WHILE NOT endMainLoop DO							
	IF left < right THEN                	
		pPivotElement										:= pCompareElement + (SizeOfStruct * TO_UDINT(SHR(right+left,1)));
		i 													:= left -1;
		j 													:= right +1;
		endSubLoop 											:= FALSE;
		REPEAT
			IF SortInverse
			THEN	// sort descending	
				REPEAT	
					i 										:= i+1;	
					pCmpElement								:= pCompareElement + (SizeOfStruct * TO_UDINT(i-1));
					FOR k := 0 TO MAX_WSTRING_LENGTH DO // Find unequal char
						// element 1,2 to upper char 	https://www.uni-due.de/hummell/infos/ascii/
						IF pCmpElement^[k] = 0 
							AND IgnoreBlank
						THEN
							CompareElement					:= 127;
						ELSE
							CompareElement					:= SEL(pCmpElement^[k] >= 97(*a*)	AND_THEN pCmpElement^[k] <= 122(*z*), 	pCmpElement^[k],pCmpElement^[k] - 32);		// a --> A
						END_IF
						IF pPivotElement^[k] = 0 
							AND IgnoreBlank
						THEN
							PivotElement					:= 127;
						ELSE
							PivotElement					:= SEL(pPivotElement^[k] >= 97(*a*) AND_THEN pPivotElement^[k] <= 122(*z*), pPivotElement^[k], 	pPivotElement^[k] - 32);// a --> A
						END_IF
						// Find unequal char
						IF CompareElement <> PivotElement
							OR CompareElement = 0
							OR PivotElement = 0
						THEN
							EXIT;
						END_IF
					END_FOR
				UNTIL (CompareElement <= PivotElement) OR NOT (i < right)	END_REPEAT	
				REPEAT	
					j 										:= j-1;	
					pCmpElement								:= pCompareElement + (SizeOfStruct * TO_UDINT(j-1));
					FOR k := 0 TO MAX_WSTRING_LENGTH DO // Find unequal char
						// element 1,2 to upper char 	https://www.uni-due.de/hummell/infos/ascii/
						IF pCmpElement^[k] = 0 
							AND IgnoreBlank
						THEN
							CompareElement					:= 127;
						ELSE
							CompareElement					:= SEL(pCmpElement^[k] >= 97(*a*)	AND_THEN pCmpElement^[k] <= 122(*z*), 	pCmpElement^[k],pCmpElement^[k] - 32);		// a --> A
						END_IF
						IF pPivotElement^[k] = 0 
							AND IgnoreBlank
						THEN
							PivotElement					:= 127;
						ELSE
							PivotElement					:= SEL(pPivotElement^[k] >= 97(*a*) AND_THEN pPivotElement^[k] <= 122(*z*), pPivotElement^[k], 	pPivotElement^[k] - 32);// a --> A
						END_IF
						// Find unequal char
						IF CompareElement <> PivotElement
							OR CompareElement = 0
							OR PivotElement = 0
						THEN
							EXIT;
						END_IF
					END_FOR
				UNTIL (CompareElement >= PivotElement) OR NOT (j > left)	END_REPEAT		
			ELSE	// sort ascending
				REPEAT	
					i 										:= i+1;
					pCmpElement								:= pCompareElement + (SizeOfStruct * TO_UDINT(i-1));
					FOR k := 0 TO MAX_WSTRING_LENGTH DO // Find unequal char
						// element 1,2 to upper char 	https://www.uni-due.de/hummell/infos/ascii/
						IF pCmpElement^[k] = 0 
							AND IgnoreBlank
						THEN
							CompareElement					:= 127;
						ELSE
							CompareElement					:= SEL(pCmpElement^[k] >= 97(*a*)	AND_THEN pCmpElement^[k] <= 122(*z*), 	pCmpElement^[k],pCmpElement^[k] - 32);		// a --> A
						END_IF
						IF pPivotElement^[k] = 0 
							AND IgnoreBlank
						THEN
							PivotElement					:= 127;
						ELSE
							PivotElement					:= SEL(pPivotElement^[k] >= 97(*a*) AND_THEN pPivotElement^[k] <= 122(*z*), pPivotElement^[k], 	pPivotElement^[k] - 32);// a --> A
						END_IF
						// Find unequal char
						IF CompareElement <> PivotElement
							OR CompareElement = 0
							OR PivotElement = 0
						THEN
							EXIT;
						END_IF
					END_FOR
				UNTIL (CompareElement >= PivotElement)	OR NOT (i < right)	END_REPEAT;				
				REPEAT	
					j 										:= j-1;	
					pCmpElement								:= pCompareElement + (SizeOfStruct * TO_UDINT(j-1));
					FOR k := 0 TO MAX_WSTRING_LENGTH DO // Find unequal char
						// element 1,2 to upper char 	https://www.uni-due.de/hummell/infos/ascii/
						IF pCmpElement^[k] = 0 
							AND IgnoreBlank
						THEN
							CompareElement					:= 127;
						ELSE
							CompareElement					:= SEL(pCmpElement^[k] >= 97(*a*)	AND_THEN pCmpElement^[k] <= 122(*z*), 	pCmpElement^[k],pCmpElement^[k] - 32);		// a --> A
						END_IF
						IF pPivotElement^[k] = 0 
							AND IgnoreBlank
						THEN
							PivotElement					:= 127;
						ELSE
							PivotElement					:= SEL(pPivotElement^[k] >= 97(*a*) AND_THEN pPivotElement^[k] <= 122(*z*), pPivotElement^[k], 	pPivotElement^[k] - 32);// a --> A
						END_IF
						// Find unequal char
						IF CompareElement <> PivotElement
							OR CompareElement = 0
							OR PivotElement = 0
						THEN
							EXIT;
						END_IF
					END_FOR
				UNTIL (CompareElement <= PivotElement) OR NOT (j > left)	END_REPEAT;
			END_IF
			IF i >= j THEN
				endSubLoop									:= TRUE;
			ELSE                    					
				Allocate(SizeOfStruct);
				pElement_1									:= pData + (SizeOfStruct * TO_UDINT(j-1));
				pElement_2									:= pData + (SizeOfStruct * TO_UDINT(i-1));
				
				IF pElement_Tmp = 0 
					OR_ELSE MEMCPY(pElement_Tmp, pElement_1,	SizeOfStruct) = 0
					OR_ELSE MEMCPY(pElement_1,	pElement_2,		SizeOfStruct) = 0
					OR_ELSE MEMCPY(pElement_2,	pElement_Tmp,	SizeOfStruct) = 0
				THEN
					byWSTRING								:= FALSE;
					RETURN;	
				END_IF

			END_IF
		UNTIL endSubLoop END_REPEAT;		
		stack[stackCount] 									:= TO_UDINT(right); 	// save right in stack			
		IF stackCount < 32              					
		THEN                            					
			stackCount 										:= stackCount +1;
		ELSE															// Error stack Limit    
			endMainLoop 									:= TRUE;
			byWSTRING										:= FALSE;			
		END_IF                          					
		right 												:= MAX(left, i-1);
	ELSE                                
		IF stackCount = 1 THEN          
			endMainLoop 									:= TRUE;
		ELSE                            					
			left 											:= right+1;       
			stackCount 										:= stackCount -1;	// load from stack
			right											:= TO_DINT(stack[stackCount]);
		END_IF
	END_IF
END_WHILE
END_METHOD

METHOD FB_exit : BOOL
VAR_INPUT
	bInCopyCode : BOOL; // if TRUE, the exit method is called for exiting an instance that is copied afterwards (online change).
END_VAR
IF NOT bInCopyCode AND pElement_Tmp <> 0
THEN //Release memory in case the PLC stopps
	__DELETE(pElement_Tmp);
END_IF
END_METHOD

END_FUNCTION_BLOCK

// POUs/EventLogger/ReadEvents/EventlogRead
{attribute 'no_check'}
//Read TwinCat ADS evenlogger messages via ADS into PLC in Unicode format
FUNCTION_BLOCK EventlogRead EXTENDS FbBase
VAR CONSTANT
	IGRP_ENUMEVENTS											: UDINT := 16#190;
	IOFFS_ENUM_CONTINUE										: UDINT := 16#1020;
	IOFFS_ENUM_CLOSE										: UDINT := 16#1030;
                                        					
	IGRP_GETTEXT											: UDINT := 16#1F4;
	IOFFS_GETCOMPLETESTRING									: UDINT := 16#0;
	IOFFS_GETSOURCENAME										: UDINT := 16#1;
                                        					
	IOFFS_BEGINENUMACTIVE									: UDINT := 16#0;
	IOFFS_BEGINENUMLOGGED									: UDINT := 16#1;
                                        	
	IGRP_TCEVENTSTREAM_SIMPLE								: UDINT := 16#1;
	IOFFS_TCEVENTCLASS_NONE 								: UDINT := 16#0;
END_VAR
VAR_OUTPUT CONSTANT
	MIN_EVENT												: INT := 1; 
	MAX_EVENT												: INT := PARAM.EVENT_HANDLING_CONFIG.EVENTLOG_READ_MAX_EVENTS ; //End index event list  - see library parameter to customize parameter
	
{attribute 'displaymode':='binary'}
	OPTION_USE_STATE_FOR_TIMESTAMP							: 	BYTE :=2#0000_0001; //option to enable timestamp according to event state instead of only signaled timestamp
{attribute 'displaymode':='binary'}
	OPTION_GET_HOSTNAME_FOR_EACH_EVENT						: 	BYTE :=2#0000_0010; //option to read host name for each single event
END_VAR                                 					
VAR_INPUT                               					
	LangId													: eLCID := eLCID.US; //See LCID 	
	NetId													: T_AMSNetId := '';
	TimeOut													: TIME := DEFAULT_ADS_TIMEOUT;
	TimezoneBias											: DINT; //Timezone bias to UTC in minutes - As timestamp provided by Evetlogger is in UTC
{attribute 'displaymode':='binary'}
	Options													: BYTE := 2#0000_0000; 
END_VAR                                 					
VAR_OUTPUT                              					
	Event													: ARRAY [MIN_EVENT..MAX_EVENT] OF EVENTLOG_READ_DATA; //Event list 
	TotalNumberOfEvents										: INT := 0; //Number of events in list
	QuitReqNumberOfEvents									: INT := 0; //Number of events in list where quit is required
	CurrentEventCount										: INT := 0; //Count down the number of events need to read 
	ExecutionTime											: TIME; //Total cycle time to read all events
	ClassStatus												: DWORD; //Overview of active TC event classes - bit number is equivalent to TcEventClass count
END_VAR
VAR
(* Local memory ********************************************)
	MemLastErrorId											:	UDINT;
	MemTargetNetId											: T_AMSNetId;
	ReadBytes												: UDINT;
	MemTimeStartCycle										: TIME;
	MemClassStatus											: DWORD;
	MemEventFiletime										: T_FILETIME;	                         					
	MemADSEvent												: EVENTLOG_READ_DATA;
	                                    					
	EventStream												: EVENTLOG_READ_STREAM;
	HandleInfo												: EVENTLOG_READ_HANDLEINFO;
	PassHandleInfo											: EVENTLOG_READ_HANDLEINFO;

	CopyLen													:	UDINT;
(* Timer *******************************************************)

(* Trigger *****************************************************)
	
(* function-blocks *********************************************)
	fbAdsRead												: ADSREAD;
	fbAdsReadWrite											: ADSRDWRTEX;
	fbAdsWrite												: ADSWRITE;
	fbGetHostName											: FB_GetHostName;
	
(* Error *******************************************************)

(* internal used dummys *************************************)
	i														: 	UINT := 0 ;
END_VAR

	(* Read Eventlogger messages via ADS into the PLC  			 Unicode	*)
	(************************************************************************)

(* action **************************************************************************)
rtExecute(CLK := Execute);
CASE State OF
	0: 	(* Begin *)
		IF rtExecute.Q
		THEN
			Busy 											:= TRUE;
			Done 											:= FALSE;
			Error 											:= FALSE;
			ErrorId 										:= 0;
			fbAdsRead(READ := FALSE);           			
			fbAdsReadWrite(WRTRD := FALSE);     			
			fbAdsWrite(WRITE := FALSE);         			
			fbGetHostName(bExecute := FALSE);   			
			MemTimeStartCycle								:= TIME();
			MemClassStatus									:= 0;
			State 											:= 1;
                                                				
		ELSIF NOT Execute                       				
		THEN                                    				
			Done											:= FALSE;
			Busy 											:= FALSE;
			Error 											:= FALSE;
			ErrorId 										:= 0;
		END_IF

	1:	(* Get Handle*)
		fbAdsRead(
			NETID		:= NetId,
			PORT		:= AMSPORT_EVENTLOG,
			IDXGRP		:= IGRP_ENUMEVENTS,
			IDXOFFS		:= 16#1000 + IOFFS_BEGINENUMACTIVE,
			LEN			:= SIZEOF(HandleInfo),
			DESTADDR	:= ADR(HandleInfo),
			READ		:= TRUE,
			TMOUT		:= Timeout,
			BUSY		=> ,
			ERR			=> ,
			ErrId		=> );

		IF NOT fbAdsRead.BUSY
		THEN
			IF NOT fbAdsRead.ERR
			THEN
				CurrentEventCount 							:= LIMIT(0,DWORD_TO_INT(HandleInfo.Count),MAX_EVENT);
				TotalNumberOfEvents 						:= CurrentEventCount;
				QuitReqNumberOfEvents						:= CurrentEventCount;
				
				IF CurrentEventCount < 1
				THEN (* no actice event *)
					MEMSET(ADR(Event),0,SIZEOF (Event)); (* alle Events loeschen *)
					state 									:= 99;
				ELSE (* start reading data - deleting rest of current list *)
					MEMSET(ADR(Event[MIN(TotalNumberOfEvents + 1,MAX_EVENT)]),0, SIZEOF(Event[1]) * TO_UDINT((MAX_EVENT - TotalNumberOfEvents)));
					
					state 									:= 2;
				END_IF
				
			ELSE
				CurrentEventCount 							:= 1;
				TotalNumberOfEvents 						:= 1;
				QuitReqNumberOfEvents						:= 1;				
				ErrorId										:= fbAdsRead.ERRID;
				MEMSET(ADR(Event),0,SIZEOF (Event)); (* alle Events loeschen *)
				Event[1].Class								:= TCEVENTCLASS_ALARM;
				Event[1].MsgText							:= WCONCAT("Error get event handle - Error ID: ", TO_WSTRING(ErrorId));
				Event[1].MegLen								:= TO_DWORD(WLEN(Event[1].MsgText));
				Event[1].Source								:= "<Unknown>";	
				Event[1].Computer							:= '<Local>';	
				
				State 										:= 99;
			END_IF
			fbAdsRead(READ := FALSE);		
		END_IF

	(* Read Event Stream **************************************************************)
	2: 
		PassHandleInfo.Enum 								:= HandleInfo.Enum;
		PassHandleInfo.Count 								:= 1;

		fbAdsReadWrite(
			NETID		:= NetId,
			PORT		:= AMSPORT_EVENTLOG,
			IDXGRP		:= IGRP_ENUMEVENTS,
			IDXOFFS		:= IOFFS_ENUM_CONTINUE,
			WRITELEN	:= SIZEOF(PassHandleInfo),
			READLEN		:= SIZEOF(EventStream),
			SRCADDR		:= ADR(PassHandleInfo),
			DESTADDR	:= ADR(EventStream),
			WRTRD		:= TRUE,
			TMOUT		:= Timeout,
			BUSY		=> ,
			ERR			=> ,
			ErrId		=> ,
			COUNT_R		=> ReadBytes);
			
		IF NOT fbAdsReadWrite.BUSY
		THEN
			IF NOT fbAdsReadWrite.ERR
			THEN
				IF EventStream.data.zFmtProgId = '' THEN
					EventStream.data.zFmtProgId 			:= 'TcEventFormatter.TcXmlFormatter';
				END_IF
				EventStream.cbStream 						:= EventStream.cbStream + 2;
				EventStream.count 							:= TO_DWORD(LangId);
				(* Target NetId from Event array *)
				MemTargetNetId 								:= F_CreateAmsNetId(EventStream.data.AdsAddr);
				
				MEMSET(ADR(MemAdsEvent),0,SIZEOF(MemAdsEvent));
					
				MemADSEvent.Class							:= DWORD_TO_UINT(EventStream.data.Class);
				MemADSEvent.id 								:= EventStream.data.Id;
				MemADSEvent.SourceId						:= EventStream.data.SrcId;
				MemADSEvent.State							:= EventStream.data.State;
				MemADSEvent.Flags							:= EventStream.data.Flags;
						
				IF NOT Options.0
				THEN
					MemADSEvent.Timestamp					:= FILETIME_TO_DCTIME64(EventStream.data.TimeSignaled);							
				ELSE
					CASE MemADSEvent.State OF
					TCEVENTSTATE_SIGNALED:	
						MemADSEvent.Timestamp				:= FILETIME_TO_DCTIME64(EventStream.data.TimeSignaled);							
					TCEVENTSTATE_RESET:									
						MemADSEvent.Timestamp				:= FILETIME_TO_DCTIME64(EventStream.data.TimeReseted);	
					TCEVENTSTATE_CONFIRMED:					
						MemADSEvent.Timestamp				:= FILETIME_TO_DCTIME64(EventStream.data.TimeConfirmed);	
					TCEVENTSTATE_RESETCON:			
						MemADSEvent.Timestamp				:= MAX(FILETIME_TO_DCTIME64(EventStream.data.TimeReseted),FILETIME_TO_DCTIME64(EventStream.data.TimeConfirmed));				
					ELSE //TCEVENTSTATE_INVALID:
						MemADSEvent.Timestamp				:= FILETIME_TO_DCTIME64(EventStream.data.TimeSignaled);	
					END_CASE					
				END_IF
				IF TimezoneBias > 0
				THEN
					MemADSEvent.Timestamp					:= MemADSEvent.Timestamp + (60 * EC_DCTIME_TICKSPERSEC64 * TO_ULINT(TimezoneBias));
				ELSIF TimezoneBias < 0
				THEN
					MemADSEvent.Timestamp					:=  MemADSEvent.Timestamp - (TO_ULINT(ABS(TimezoneBias)) * 60 * EC_DCTIME_TICKSPERSEC64);
				END_IF
				MemADSEvent.TimestampDT						:= FILETIME_TO_DT(DCTIME64_TO_FILETIME(MemADSEvent.Timestamp));	
				MemClassStatus								:= SETBIT32(MemClassStatus, UINT_TO_SINT(Event[CurrentEventCount].Class));
				state 										:= 3;
			ELSE
				ErrorId 									:= fbAdsReadWrite.ErrId;
				MEMSET(ADR(MemTargetNetId),0,SIZEOF(MemTargetNetId));
				MEMSET(ADR(MemAdsEvent),0,SIZEOF(MemAdsEvent));	
				MemADSEvent.Class							:= TCEVENTCLASS_ALARM;				
				MemADsEvent.MsgText							:= WCONCAT("Error read event stream - Error ID: ", TO_WSTRING(ErrorId));
				MemADsEvent.MegLen							:= TO_DWORD(WLEN(MemADsEvent.MsgText));
				EventStream.count 							:= TO_DWORD(LangId);
				MemClassStatus								:= SETBIT32(MemClassStatus, UINT_TO_SINT(Event[CurrentEventCount].Class));
				state 										:= 4;				
			END_IF
			
			fbAdsReadWrite(WRTRD := FALSE);		

		END_IF

	3:	(* Read Msg Text *)
		fbAdsReadWrite(
			NETID		:= NetId,
			PORT		:= AMSPORT_EVENTLOG,
			IDXGRP		:= IGRP_GETTEXT,
			IDXOFFS		:= IOFFS_GETCOMPLETESTRING,
			WRITELEN	:= EventStream.cbStream ,
			READLEN		:= SIZEOF(EventStream.data.evtData.Temp),
			SRCADDR		:= ADR(EventStream),
			DESTADDR	:= ADR(EventStream.data.evtData.Temp),
			WRTRD		:= TRUE,
			TMOUT		:= Timeout,
			BUSY		=> ,
			ERR			=> ,
			ErrId		=> ,
			COUNT_R		=> ReadBytes);

		IF NOT fbAdsReadWrite.BUSY
		THEN
			IF NOT fbAdsReadWrite.ERR
			THEN
				//Use unicode
				CopyLen										:= MIN(ReadBytes, SIZEOF(MemADsEvent.MsgText) - 2);
				MEMCPY(ADR(MemADsEvent.MsgText),ADR(EventStream.data.evtData.Temp),CopyLen);
				MemADsEvent.MegLen							:= CopyLen;
				MemADsEvent.MsgText[CopyLen]				:= 0; 
				
				state 										:= 4;
			ELSE
				ErrorId 									:= fbAdsReadWrite.ErrId;
				MemADsEvent.MsgText							:= WCONCAT("Error read event message - Error ID: ", TO_WSTRING(ErrorId));
				MemADsEvent.MegLen							:= TO_DWORD(WLEN(MemADsEvent.MsgText));
				State 										:= 4;
			END_IF
			fbAdsReadWrite(WRTRD := FALSE);		

		END_IF

	4:	(* Read Source Name *)
		PassHandleInfo.Enum 								:= HandleInfo.Enum;
		PassHandleInfo.Count 								:= 1;

		fbAdsReadWrite(
			NETID		:= NetId,
			PORT		:= AMSPORT_EVENTLOG,
			IDXGRP		:= IGRP_GETTEXT,
			IDXOFFS		:= IOFFS_GETSOURCENAME,
			WRITELEN	:= EventStream.cbStream,
			READLEN		:= SIZEOF(EventStream.data.evtData.Temp),
			SRCADDR		:= ADR(EventStream),
			DESTADDR	:= ADR(EventStream.data.evtData.Temp),
			WRTRD		:= TRUE,
			TMOUT		:= Timeout,
			BUSY		=> ,
			ERR			=> ,
			ErrId		=> ,
			COUNT_R		=> ReadBytes);

		IF NOT fbAdsReadWrite.BUSY
		THEN
			IF NOT fbAdsReadWrite.ERR
			THEN
				CopyLen										:= MIN(ReadBytes, SIZEOF(MemADsEvent.Source) - 2);
				MEMCPY(ADR(MemADsEvent.Source),ADR(EventStream.data.evtData.Temp),CopyLen);						
		
			ELSIF fbAdsReadWrite.ErrId = 16#80070057 OR  fbAdsReadWrite.ErrId = 16#80030002
			THEN
				MemAdsEvent.Source							:= WCONCAT("Name unknown id ", TO_WSTRING(EventStream.data.SrcId));
			ELSE
				ErrorId 									:= fbAdsReadWrite.ErrId;
				MemAdsEvent.Source				 			:= "<Unknown>";
			END_IF
		
			state											:= 5;
			fbAdsReadWrite(WRTRD := FALSE);		

		END_IF
		
	5: (* Read Host Name *)
		fbGetHostName(
			sNetID		:= MemTargetNetId ,
			bExecute	:= fbGetHostName.sHostName <> '' OR Options.1,
			tTimeout	:= Timeout,
			bBusy		=> ,
			bError		=> ,
			nErrId		=> ,
			sHostName	=> );

		IF NOT fbGetHostName.bBusy
		THEN
			IF fbGetHostName.bError
			THEN
				MemAdsEvent.Computer						:= '<Unknown>';
			ELSE
				MemAdsEvent.Computer						:= fbGetHostName.sHostName;		
			END_IF

			//Copy event to 
			Event[CurrentEventCount]						:= MemAdsEvent;	
	
			//Count quit required events 
			IF NOT MemAdsEvent.Flags.1
			THEN
				QuitReqNumberOfEvents						:= QuitReqNumberOfEvents - 1;
			END_IF
					
			(* other messages *)
			CurrentEventCount 								:= CurrentEventCount - 1;
			IF CurrentEventCount < 1 THEN
				state 										:= 99;
			ELSE
				state 										:= 2;
			END_IF
			
			fbGetHostName(bExecute := FALSE);
		END_IF

	99: 	(* Close *)				
		fbAdsWrite(
			NETID	:= NetId,
			PORT	:= AMSPORT_EVENTLOG,
			IDXGRP	:= IGRP_ENUMEVENTS,
			IDXOFFS	:= IOFFS_ENUM_CLOSE,
			LEN		:= SIZEOF(HandleInfo.Enum),
			SRCADDR	:= ADR(HandleInfo),
			WRITE	:= state = 99,
			TMOUT	:= Timeout,
			BUSY	=> ,
			ERR		=> ,
			ErrId	=> );

		IF NOT fbAdsWrite.BUSY
		THEN
			ExecutionTime	 								:= TIME() - MemTimeStartCycle;
			Done											:= ErrorId = 0 AND Busy;
			Error 											:= NOT Done;
			ErrorId 										:= SEL(fbAdsWrite.ERR, ErrorId,fbAdsWrite.ErrId);
			MemLastErrorid									:= ErrorId;
			ClassStatus										:= MemClassStatus;
			Busy 											:= FALSE;
			State 											:= 0;

			fbAdsWrite(WRITE := FALSE);
		END_IF

	END_CASE
	
(*************************************************************************************************)

PROPERTY PUBLIC optGetHostNameForEachEvent : bool
GET
optGetHostNameForEachEvent := Options.1;
END_GET
SET
Options.1 := optGetHostNameForEachEvent;
END_SET
END_PROPERTY

PROPERTY PUBLIC optUseStateForTimestamp : bool
GET
optUseStateForTimestamp := Options.0;
END_GET
SET
Options.0 := optUseStateForTimestamp;
END_SET
END_PROPERTY

END_FUNCTION_BLOCK

// POUs/EventLogger/TriggerEvents/EventHandling
{attribute 'no_check'}
//ADSLOGEVENT wrapper for a convenient and pre configured use - see Beckhoff documentation for more information about AdsEventLogger
//See Param constanst to configure whether the TcEventClass need to be acknowledged (confirmation required) 
FUNCTION_BLOCK EventHandling
VAR_INPUT
	Flag													:	BOOL := FALSE; //Fire event 
	ConfirmTrig												:	BOOL := FALSE; //Ack event
	MsgId													:	UINT := 0; //Event number
	SourceId												: 	UDINT:= 0; //Event source number
	eClass													:	E_TcEventClass := TCEVENTCLASS_ALARM; (*	TC2_SYSTEM.TCEVENTCLASS_NONE		
																											TC2_SYSTEM.TCEVENTCLASS_MAINTENANCE
																											TC2_SYSTEM.TCEVENTCLASS_MESSAGE		
																											TC2_SYSTEM.TCEVENTCLASS_HINT		
																											TC2_SYSTEM.TCEVENTCLASS_STATEINFO	
																											TC2_SYSTEM.TCEVENTCLASS_INSTRUCTION	
																											TC2_SYSTEM.TCEVENTCLASS_WARNING		
																											TC2_SYSTEM.TCEVENTCLASS_ALARM		
																											TC2_SYSTEM.TCEVENTCLASS_PARAMERROR	*)

	Text1													:	STRING(20) := ''; //Short info text with lenght 20 chars 
	Text2													:	STRING(40) := ''; //Long info text with lenght 40 chars
	pText3													:	POINTER TO STRING := 0; //Pointer to extended info text 
END_VAR
VAR_OUTPUT
{attribute 'displaymode':='hex'}
	State													:	UDINT ; (*	TCEVENTSTATE_INVALID  	: WORD := 16#0000; 		
																			TCEVENTSTATE_SIGNALED  	: WORD := 16#0001; 		- The event is signaled 
																			TCEVENTSTATE_RESET  	: WORD := 16#0002; 		- The event is gone 
																			TCEVENTSTATE_CONFIRMED  : WORD := 16#0010 (16); - The event is confirmed 
																			TCEVENTSTATE_RESETCON  	: WORD := 16#0012 (18); - The event is gone AND confirmed *)
{attribute 'displaymode':='binary'}
	Status													:	DWORD; (*	.0 - .8 = event <class id>  / .15 confirm required / .16 = Level 0 , .17 = Level 1 , .18 = Level 2, .......... / .31 active
																			TCEVENTCLASS_NONE			:=0,
																			TCEVENTCLASS_MAINTENANCE	:=1,
																			TCEVENTCLASS_MESSAGE		:=2,
																			TCEVENTCLASS_HINT			:=3,
																			TCEVENTCLASS_STATEINFO		:=4, 
																			TCEVENTCLASS_INSTRUCTION	:=5,
																			TCEVENTCLASS_WARNING		:=6,
																			TCEVENTCLASS_ALARM			:=7,
																			TCEVENTCLASS_PARAMERROR		:=8	 *)
END_VAR
VAR
	format													:	STRING(6) := '%s%s%s';
	pPara													:	ARRAY[1..3] OF POINTER TO BYTE;
	TmpString												:	STRING(1) := '';
	AdsEvent												:	ADSLOGEVENT :=(
																	NETID				:= '',
																	PORT				:= AMSPORT_EVENTLOG,
																	TMOUT 				:= DEFAULT_ADS_TIMEOUT,
																	EventDataLength		:= 0,	
																	EventConfigData 	:= (
																		Class 				:= TCEVENTCLASS_ALARM,
																		Prio 				:= TCEVENTPRIO_IMPLICIT,
																		ProgId 				:= 'TcEventFormatter.TcXmlFormatter',
																		Flags 				:= TCEVENTFLAG_LOG OR TCEVENTFLAG_SRCID, // 16#0140 (* T *),
																		StreamType 			:= TCEVENTSTREAM_SIMPLE (* TCEVENTSTREAM_NORMAL *),
																		bQuitRequired 		:= TRUE));
END_VAR

(* EventHandling including textinfos which are send to the eventlogger  	v4.3	*)
(* specific eventclasses have to be quit, see Param.EventConfig...					*)
(************************************************************************************)

(* sequence *************************************************************)
	IF Status.31 //Message active
	THEN (* work EventLogger *)
		AdsEvent(
			NETID			:= ,(* see declaration *)
			PORT			:= ,(* see declaration *)
			Event			:= NOT AdsEvent.FbCleanup AND(Flag OR AdsEvent.EventState = TCEVENTSTATE_INVALID AND NOT AdsEvent.Quit), (* Set Event until state <> invalid *)
			EventQuit		:= AdsEvent.EventState <> TCEVENTSTATE_INVALID
								AND AdsEvent.EventConfigData.bQuitRequired
								AND NOT AdsEvent.Eventstate.4 //confirmed
								AND NOT AdsEvent.Quit
								AND(
								ConfirmTrig
								OR AdsEvent.EventQuit), (* quit send *)
			EventConfigData	:= ,(* see declaration *)
			EventDataAddress:= ADR(pPara),
			EventDataLength	:= ,(* see declaration *)
			FbCleanup		:= NOT AdsEvent.FbCleanup AND(AdsEvent.Err OR AdsEvent.EventState = TCEVENTSTATE_RESETCON),
			TMOUT			:= ,(* see declaration *)
			EventState		=> ,
			Err				=> ,
			ErrId			=> ,
			Quit			=> );
			
		IF AdsEvent.Event 
			AND AdsEvent.EventState = TCEVENTSTATE_INVALID
		THEN
			State 											:= SEL(Flag, TCEVENTSTATE_RESET, TCEVENTSTATE_SIGNALED);
		ELSIF AdsEvent.Quit
			AND AdsEvent.EventState = TCEVENTSTATE_INVALID
			AND AdsEvent.EventQuit
			OR 
			AdsEvent.FbCleanup		
		THEN
			State 											:= TCEVENTSTATE_RESETCON;
		ELSIF(AdsEvent.Err OR NOT AdsEvent.Event AND AdsEvent.EventState = TCEVENTSTATE_INVALID)
			AND_THEN Gvl.EventHandlingStatistic.CountOut(Status)
		THEN
			State											:= TCEVENTSTATE_INVALID;
		ELSE
			State											:= MAX(State, AdsEvent.EventState);
		END_IF
			
	ELSIF Flag AND SourceId > 0 
	THEN (* fire event *)
		IF PARAM.EVENT_HANDLING_CONFIG.ENABLE_DYNAMIC_EVENT_MSG_FORMAT
		THEN
			IF pText3 <> 0 AND_THEN pText3^[0] > 0
			THEN 
				format 										:= '%s%s%s'; 
			ELSIF Text2[0] > 0 
			THEN 
				format 										:= '%s%s';
			ELSIF Text1[0] > 0 
			THEN 												
				format 										:= '%s';
			ELSE
				format 										:= '';
			END_IF
		END_IF
							 
		AdsEvent.EventConfigData.DataFormatStrAddress		:= ADR(format);
		AdsEvent.EventConfigData.Id 						:= UINT_TO_UDINT(MsgID);
		AdsEvent.EventConfigData.SourceId 					:= SourceId;
		Status												:= Gvl.EventHandlingStatistic.InitEvent(SetClass := eClass, EventConfig := AdsEvent.EventConfigData);		

		(* Data *)
		pPara[1] 											:= ADR(Text1);
		pPara[2] 											:= ADR(Text2);
		pPara[3] 											:= SEL(pText3 <> 0,ADR(TmpString) ,pText3);
	
		IF AdsEvent.Err AND NOT AdsEvent.FbCleanup
		THEN
			AdsEvent(
				Event			:= FALSE,
				EventQuit 		:= FALSE,
				EventDataAddress:= ADR(pPara),
				FbCleanup		:= TRUE,
				EventState		=> );
				
		ELSE (* Fire Event *)
			AdsEvent( 	
				Event			:= FALSE,
				EventQuit 		:= FALSE, 
				FbCleanup 		:= FALSE, 
				EventDataAddress:= ADR(pPara));
						
			AdsEvent( 	Event 	:= TRUE);
			IF NOT AdsEvent.Err AND_THEN Gvl.EventHandlingStatistic.CountIn(Status) //Add event to statistic and continue if added successfully
			THEN			
				State 										:= TCEVENTSTATE_SIGNALED;
			END_IF
						
		END_IF
	END_IF

(**********************************************************************************)

END_FUNCTION_BLOCK

// POUs/EventLogger/TriggerEvents/EventHandlingConfirmIsReq
{attribute 'no_check'}
//Returns status of "QuitRequired" configuration for corresponding event class (see library Param) 
FUNCTION EventHandlingConfirmIsReq : BOOL
VAR_INPUT
	TcEventClass											:	E_TcEventClass;
END_VAR
VAR
END_VAR

	CASE tcEventClass OF
	Tc2_System.TCEVENTCLASS_NONE:			EventHandlingConfirmIsReq	:= PARAM.EVENT_HANDLING_CONFIG.CLASS_NONE_QUIT_REQUIRED;	
	Tc2_System.TCEVENTCLASS_MAINTENANCE:	EventHandlingConfirmIsReq	:= PARAM.EVENT_HANDLING_CONFIG.CLASS_MAINTENANCE_QUIT_REQUIRED;		
	Tc2_System.TCEVENTCLASS_MESSAGE:		EventHandlingConfirmIsReq	:= PARAM.EVENT_HANDLING_CONFIG.CLASS_MESSAGE_QUIT_REQUIRED;			
	Tc2_System.TCEVENTCLASS_HINT:			EventHandlingConfirmIsReq	:= PARAM.EVENT_HANDLING_CONFIG.CLASS_HINT_QUIT_REQUIRED;	
	Tc2_System.TCEVENTCLASS_STATEINFO:		EventHandlingConfirmIsReq	:= PARAM.EVENT_HANDLING_CONFIG.CLASS_STATEINFO_QUIT_REQUIRED;	
	Tc2_System.TCEVENTCLASS_INSTRUCTION:	EventHandlingConfirmIsReq	:= PARAM.EVENT_HANDLING_CONFIG.CLASS_INSTRUCTION_QUIT_REQUIRED;	
	Tc2_System.TCEVENTCLASS_WARNING:		EventHandlingConfirmIsReq	:= PARAM.EVENT_HANDLING_CONFIG.CLASS_WARNING_QUIT_REQUIRED;	
	Tc2_System.TCEVENTCLASS_ALARM:			EventHandlingConfirmIsReq	:= PARAM.EVENT_HANDLING_CONFIG.CLASS_ALARM_QUIT_REQUIRED;	
	Tc2_System.TCEVENTCLASS_PARAMERROR:		EventHandlingConfirmIsReq	:= PARAM.EVENT_HANDLING_CONFIG.CLASS_PARAMERROR_QUIT_REQUIRED;		
	ELSE                                                    
		EventHandlingConfirmIsReq										:= PARAM.EVENT_HANDLING_CONFIG.CLASS_ALARM_QUIT_REQUIRED;
	END_CASE

END_FUNCTION

// POUs/EventLogger/TriggerEvents/EventHandlingGrp10
{attribute 'no_check'}
//Event group with single source id - for a convenient control of <MAX_EVENTS>
//Each single event handling FB is accessible, so that signal flag, information text and alarm class could be used
FUNCTION_BLOCK EventHandlingGrp10
VAR_OUTPUT CONSTANT
	MIN_EVENT												:	INT := 1; 
	MAX_EVENT												:	INT := 10;
END_VAR                                                 	
VAR_INPUT                                               	
	ConfirmTrig												:	BOOL := FALSE; //Acknowledge event
	SourceId												: 	UDINT := 0; //Source id for all events of this group
	no														:	ARRAY [MIN_EVENT..MAX_EVENT] OF EventHandling; //Array of single event handling FBs 
	Disable													:	BOOL := FALSE; //Disable all events 
	AutoConfirm												:	BOOL := FALSE; //All events will be acknowledged if flag is gone *)
	SetClass												:	E_TcEventClass := TC2_SYSTEM.TCEVENTCLASS_ALARM;// if set class is <> ALARM -> all events set to this Eventclass
	MsgOffset												:	INT := 0; //Offset to change default message id to MIN_EVENT to MsgOffset
END_VAR                                                 	
VAR_OUTPUT    
{attribute 'displaymode':='binary'}
	Status													:	DWORD; (*	.0 - .8 = event of <class id> is active / .15 confirm required / .16 = Level 0 , .17 = Level 1 , .18 = Level 2, ..........
																			TCEVENTCLASS_NONE			:=0,	(* No class *)
																			TCEVENTCLASS_MAINTENANCE	:=1,	(* Maintenance hint *)
																			TCEVENTCLASS_MESSAGE		:=2,	(* Message *)
																			TCEVENTCLASS_HINT			:=3,	(* Hint *)
																			TCEVENTCLASS_STATEINFO		:=4,	(* State information *)
																			TCEVENTCLASS_INSTRUCTION	:=5,	(* Instruction *)
																			TCEVENTCLASS_WARNING		:=6,	(* Warning *)
																			TCEVENTCLASS_ALARM			:=7,	(* Alarm *)
																			TCEVENTCLASS_PARAMERROR		:=8		(* Parameter error *)  *)
	NoOfActiveEvents										:	INT;
END_VAR                                                 	
VAR                                                     	
	_Mem													:	BYTE;
	Disabled												:	BOOL;
	i 														:	INT;
END_VAR

(* EventHandlingGrp			V4.1	*)
(************************************)

(* status ***************************)
Status  													:= 0;
NoOfActiveEvents											:= 0;

IF(Disable OR SourceId = 0)AND Disabled
THEN
	RETURN;
ELSE	
	Disabled												:= Disable OR SourceId = 0;
	
	FOR i := MIN_EVENT TO MAX_EVENT 
	DO
		(* Init Default Class *)
		IF SetClass <> TC2_SYSTEM.TCEVENTCLASS_ALARM
			AND NOT _Mem.7
		THEN
			no[i].eClass										:= SetClass;
			_Mem.7											:= i = MAX_EVENT;
		END_IF                                  			
		                                        			
		IF Disable OR SourceId = 0              			
		THEN                                    			
			no[i].Flag 										:= FALSE;
			no[i].ConfirmTrig 								:= no[i].State <> TCEVENTSTATE_INVALID AND no[i].State <> TCEVENTSTATE_RESETCON;
		ELSIF ConfirmTrig                             			
		THEN                                    	
			no[i].ConfirmTrig 								:= TRUE;
			_Mem.0 											:= ConfirmTrig;
                                                			
		ELSIF _Mem.0                            			
		THEN                                    			
			no[i].ConfirmTrig 								:= FALSE;
			_Mem.0 											:= i <> MAX_EVENT;

		ELSIF AutoConfirm
		THEN
			IF NOT no[i].Flag
				AND no[i].State <> TCEVENTSTATE_INVALID
				AND no[i].State <> TCEVENTSTATE_RESETCON
			THEN
				no[i].ConfirmTrig 							:= TRUE;
			ELSE                                			
				no[i].ConfirmTrig 							:= FALSE;
			END_IF                              			
		END_IF                                  	
                                                	
		(* Mem current Event *)                 	
		IF no[i].State <> TCEVENTSTATE_INVALID OR no[i].Flag 
		THEN
			_Mem.1											:= TRUE;
			(* Call Event *)
			no[i](
				Flag	:= ,
				ConfirmTrig := ,
				MsgId	:= TO_UINT(i + MsgOffset),
				SourceId:= SourceId,
				eClass	:= (* see grp call *),
				Text1	:= (* see grp call *),
				Text2	:= (* see grp call *),
				pText3	:= (* see grp call *),
				State	=> );
		END_IF

		(* Set info flags *)
		IF	no[i].State <> TCEVENTSTATE_INVALID 
		THEN
			NoOfActiveEvents								:= NoOfActiveEvents + 1;
			Status											:= Status OR no[i].Status;
			Disabled										:= FALSE;
		ELSIF _Mem.1
		THEN (* Send one time info event is gone *)
			; 
		END_IF
	END_FOR	
END_IF
(*****************************************************************************************)

METHOD PUBLIC confirm : booL //Return value = TRUE if execution finished
VAR_INPUT
END_VAR
IF NoOfActiveEvents > 0
THEN
	FOR i := MIN_EVENT TO MAX_EVENT 
	DO
		no[i](ConfirmTrig := TRUE);
	END_FOR
	_Mem.0			:= TRUE;
END_IF

confirm		:= TRUE;
END_METHOD

PROPERTY PUBLIC confirmIsReq : BOOL
GET
confirmIsReq							:= Status.15;
END_GET
END_PROPERTY

PROPERTY PUBLIC isActive : BOOL
GET
IsActive 								:= Status <> 0;
END_GET
END_PROPERTY

END_FUNCTION_BLOCK

// POUs/EventLogger/TriggerEvents/EventHandlingGrp25
{attribute 'no_check'}
//Event group with single source id - for a convenient control of <MAX_EVENTS>
//Each single event handling FB is accessible, so that signal flag, information text and alarm class could be used
FUNCTION_BLOCK EventHandlingGrp25
VAR_OUTPUT CONSTANT
	MIN_EVENT												:	INT := 1; 
	MAX_EVENT												:	INT := 25;
END_VAR                                                 	
VAR_INPUT                                               	
	ConfirmTrig												:	BOOL := FALSE; //Acknowledge event
	SourceId												: 	UDINT := 0; //Source id for all events of this group
	no														:	ARRAY [MIN_EVENT..MAX_EVENT] OF EventHandling; //Array of single event handling FBs 
	Disable													:	BOOL := FALSE; //Disable all events 
	AutoConfirm												:	BOOL := FALSE; //All events will be acknowledged if flag is gone *)
	SetClass												:	E_TcEventClass := TC2_SYSTEM.TCEVENTCLASS_ALARM;// if set class is <> ALARM -> all events set to this Eventclass
	MsgOffset												:	INT := 0; //Offset to change default message id to MIN_EVENT to MsgOffset
END_VAR                                                 	
VAR_OUTPUT    
{attribute 'displaymode':='binary'}
	Status													:	DWORD; (*	.0 - .8 = event of <class id> is active / .15 confirm required / .16 = Level 0 , .17 = Level 1 , .18 = Level 2, ..........
																			TCEVENTCLASS_NONE			:=0,	(* No class *)
																			TCEVENTCLASS_MAINTENANCE	:=1,	(* Maintenance hint *)
																			TCEVENTCLASS_MESSAGE		:=2,	(* Message *)
																			TCEVENTCLASS_HINT			:=3,	(* Hint *)
																			TCEVENTCLASS_STATEINFO		:=4,	(* State information *)
																			TCEVENTCLASS_INSTRUCTION	:=5,	(* Instruction *)
																			TCEVENTCLASS_WARNING		:=6,	(* Warning *)
																			TCEVENTCLASS_ALARM			:=7,	(* Alarm *)
																			TCEVENTCLASS_PARAMERROR		:=8		(* Parameter error *)  *)
	NoOfActiveEvents										:	INT;																		
END_VAR                                                 	
VAR                                                     	
	_Mem													:	BYTE;
	Disabled												:	BOOL;
	i 														:	INT;
END_VAR

(* EventHandlingGrp			V4.1	*)
(************************************)

(* status ***************************)
Status  													:= 0;
NoOfActiveEvents											:= 0;

IF(Disable OR SourceId = 0)AND Disabled
THEN
	RETURN;
ELSE
	Disabled												:= Disable OR SourceId = 0;
	
	FOR i := MIN_EVENT TO MAX_EVENT 
	DO
		(* Init Default Class *)
		IF SetClass <> TC2_SYSTEM.TCEVENTCLASS_ALARM
			AND NOT _Mem.7
		THEN
			no[i].eClass										:= SetClass;
			_Mem.7											:= i = MAX_EVENT;
		END_IF                                  			
		                                        			
		IF Disable OR SourceId = 0              			
		THEN                                    			
			no[i].Flag 										:= FALSE;
			no[i].ConfirmTrig 								:= no[i].State <> TCEVENTSTATE_INVALID AND no[i].State <> TCEVENTSTATE_RESETCON;
		ELSIF ConfirmTrig                             			
		THEN                                    	
			no[i].ConfirmTrig 								:= TRUE;
			_Mem.0 											:= ConfirmTrig;
                                                			
		ELSIF _Mem.0                            			
		THEN                                    			
			no[i].ConfirmTrig 								:= FALSE;
			_Mem.0 											:= i <> MAX_EVENT;

		ELSIF AutoConfirm
		THEN
			IF NOT no[i].Flag
				AND no[i].State <> TCEVENTSTATE_INVALID
				AND no[i].State <> TCEVENTSTATE_RESETCON
			THEN
				no[i].ConfirmTrig 							:= TRUE;
			ELSE                                			
				no[i].ConfirmTrig 							:= FALSE;
			END_IF                              			
		END_IF                                  	
                                                	
		(* Mem current Event *)                 	
		IF no[i].State <> TCEVENTSTATE_INVALID OR no[i].Flag 
		THEN
			_Mem.1											:= TRUE;
			(* Call Event *)
			no[i](
				Flag	:= ,
				ConfirmTrig := ,
				MsgId	:= TO_UINT(i + MsgOffset),
				SourceId:= SourceId,
				eClass	:= (* see grp call *),
				Text1	:= (* see grp call *),
				Text2	:= (* see grp call *),
				pText3	:= (* see grp call *),
				State	=> );
		END_IF

		(* Set info flags *)
		IF	no[i].State <> TCEVENTSTATE_INVALID 
		THEN
			NoOfActiveEvents								:= NoOfActiveEvents + 1;
			Status											:= Status OR no[i].Status;
			Disabled										:= FALSE;
		ELSIF _Mem.1
		THEN (* Send one time info event is gone *)
			; 
		END_IF
	END_FOR	
END_IF
(*****************************************************************************************)

METHOD PUBLIC confirm : booL //Return value = TRUE if execution finished
VAR_INPUT
END_VAR
IF NoOfActiveEvents > 0
THEN
	FOR i := MIN_EVENT TO MAX_EVENT 
	DO
		no[i](ConfirmTrig := TRUE);
	END_FOR
	_Mem.0			:= TRUE;
END_IF

confirm		:= TRUE;
END_METHOD

PROPERTY PUBLIC confirmIsReq : BOOL
GET
confirmIsReq							:= Status.15;
END_GET
END_PROPERTY

PROPERTY PUBLIC isActive : BOOL
GET
IsActive 								:= Status <> 0;
END_GET
END_PROPERTY

END_FUNCTION_BLOCK

// POUs/EventLogger/TriggerEvents/EventHandlingGrp50
{attribute 'no_check'}
//Event group with single source id - for a convenient control of <MAX_EVENTS>
//Each single event handling FB is accessible, so that signal flag, information text and alarm class could be used
FUNCTION_BLOCK EventHandlingGrp50
VAR_OUTPUT CONSTANT
	MIN_EVENT												:	INT := 1; 
	MAX_EVENT												:	INT := 50;
END_VAR                                                 	
VAR_INPUT                                               	
	ConfirmTrig												:	BOOL := FALSE; //Acknowledge event
	SourceId												: 	UDINT := 0; //Source id for all events of this group
	no														:	ARRAY [MIN_EVENT..MAX_EVENT] OF EventHandling; //Array of single event handling FBs 
	Disable													:	BOOL := FALSE; //Disable all events 
	AutoConfirm												:	BOOL := FALSE; //All events will be acknowledged if flag is gone *)
	SetClass												:	E_TcEventClass := TC2_SYSTEM.TCEVENTCLASS_ALARM;// if set class is <> ALARM -> all events set to this Eventclass
	MsgOffset												:	INT := 0; //Offset to change default message id to MIN_EVENT to MsgOffset
END_VAR                                                 	
VAR_OUTPUT    
{attribute 'displaymode':='binary'}
	Status													:	DWORD; (*	.0 - .8 = event of <class id> is active / .15 confirm required / .16 = Level 0 , .17 = Level 1 , .18 = Level 2, ..........
																			TCEVENTCLASS_NONE			:=0,	(* No class *)
																			TCEVENTCLASS_MAINTENANCE	:=1,	(* Maintenance hint *)
																			TCEVENTCLASS_MESSAGE		:=2,	(* Message *)
																			TCEVENTCLASS_HINT			:=3,	(* Hint *)
																			TCEVENTCLASS_STATEINFO		:=4,	(* State information *)
																			TCEVENTCLASS_INSTRUCTION	:=5,	(* Instruction *)
																			TCEVENTCLASS_WARNING		:=6,	(* Warning *)
																			TCEVENTCLASS_ALARM			:=7,	(* Alarm *)
																			TCEVENTCLASS_PARAMERROR		:=8		(* Parameter error *)  *)
	NoOfActiveEvents										:	INT;
END_VAR                                                 	
VAR                                                     	
	_Mem													:	BYTE;
	Disabled												:	BOOL;
	i 														:	INT;
END_VAR

(* EventHandlingGrp			V4.1	*)
(************************************)

(* status ***************************)
Status  													:= 0;
NoOfActiveEvents											:= 0;

IF(Disable OR SourceId = 0)AND Disabled
THEN
	RETURN;
ELSE
	Disabled												:= Disable OR SourceId = 0;
	
	FOR i := MIN_EVENT TO MAX_EVENT 
	DO
		(* Init Default Class *)
		IF SetClass <> TC2_SYSTEM.TCEVENTCLASS_ALARM
			AND NOT _Mem.7
		THEN
			no[i].eClass										:= SetClass;
			_Mem.7											:= i = MAX_EVENT;
		END_IF                                  			
		                                        			
		IF Disable OR SourceId = 0              			
		THEN                                    			
			no[i].Flag 										:= FALSE;
			no[i].ConfirmTrig 								:= no[i].State <> TCEVENTSTATE_INVALID AND no[i].State <> TCEVENTSTATE_RESETCON;
		ELSIF Confirmtrig                             			
		THEN                                    	
			no[i].ConfirmTrig 								:= TRUE;
			_Mem.0 											:= Confirmtrig;
                                                			
		ELSIF _Mem.0                            			
		THEN                                    			
			no[i].ConfirmTrig 								:= FALSE;
			_Mem.0 											:= i <> MAX_EVENT;

		ELSIF AutoConfirm
		THEN
			IF NOT no[i].Flag
				AND no[i].State <> TCEVENTSTATE_INVALID
				AND no[i].State <> TCEVENTSTATE_RESETCON
			THEN
				no[i].ConfirmTrig 							:= TRUE;
			ELSE                                			
				no[i].ConfirmTrig 							:= FALSE;
			END_IF                              			
		END_IF                                  	
                                                	
		(* Mem current Event *)                 	
		IF no[i].State <> TCEVENTSTATE_INVALID OR no[i].Flag 
		THEN
			_Mem.1											:= TRUE;
			(* Call Event *)
			no[i](
				Flag	:= ,
				ConfirmTrig := ,
				MsgId	:= TO_UINT(i + MsgOffset),
				SourceId:= SourceId,
				eClass	:= (* see grp call *),
				Text1	:= (* see grp call *),
				Text2	:= (* see grp call *),
				pText3	:= (* see grp call *),
				State	=> );
		END_IF

		(* Set info flags *)
		IF	no[i].State <> TCEVENTSTATE_INVALID 
		THEN
			NoOfActiveEvents								:= NoOfActiveEvents + 1;
			Status											:= Status OR no[i].Status;
			Disabled										:= FALSE;
		ELSIF _Mem.1
		THEN (* Send one time info event is gone *)
			; 
		END_IF
	END_FOR	
END_IF
(*****************************************************************************************)

METHOD PUBLIC confirm : booL  //Return value = TRUE if execution finished
VAR_INPUT
END_VAR
IF NoOfActiveEvents > 0
THEN
	FOR i := MIN_EVENT TO MAX_EVENT 
	DO
		no[i](ConfirmTrig := TRUE);
	END_FOR
	_Mem.0			:= TRUE;
END_IF

confirm		:= TRUE;
END_METHOD

PROPERTY PUBLIC confirmIsReq : BOOL
GET
confirmIsReq							:= Status.15;
END_GET
END_PROPERTY

PROPERTY PUBLIC isActive : BOOL
GET
IsActive 								:= Status <> 0;
END_GET
END_PROPERTY

END_FUNCTION_BLOCK

// POUs/EventLogger/TriggerEvents/EventHandlingGrpCustomized
{attribute 'no_check'}
//Event group with single source id - for a convenient control of <MAX_EVENTS>
//Each single event handling FB is accessible, so that signal flag, information text and alarm class could be used
FUNCTION_BLOCK EventHandlingGrpCustomized
VAR_OUTPUT CONSTANT
	MIN_EVENT												:	INT := 1; 
	MAX_EVENT												:	INT := PARAM.EVENT_HANDLING_CONFIG.GRP_CUSTOMISED_MAX_EVENT; //Start index no of events - see library parameter to customize parameter
END_VAR                                                 	
VAR_INPUT                                               	
	ConfirmTrig												:	BOOL := FALSE; //Acknowledge event
	SourceId												: 	UDINT := 0; //Source id for all events of this group
	no														:	ARRAY [MIN_EVENT..MAX_EVENT] OF EventHandling; //Array of single event handling FBs 
	Disable													:	BOOL := FALSE; //Disable all events 
	AutoConfirm												:	BOOL := FALSE; //All events will be acknowledged if flag is gone *)
	SetClass												:	E_TcEventClass := TC2_SYSTEM.TCEVENTCLASS_ALARM;// if set class is <> ALARM -> all events set to this Eventclass
	MsgOffset												:	INT := 0; //Offset to change default message id to MIN_EVENT to MsgOffset
END_VAR                                                 	
VAR_OUTPUT                                              	
{attribute 'displaymode':='binary'}
	Status													:	DWORD; (*	.0 - .8 = event of <class id> is active / .15 confirm required / .16 = Level 0 , .17 = Level 1 , .18 = Level 2, ..........
																			TCEVENTCLASS_NONE			:=0,	(* No class *)
																			TCEVENTCLASS_MAINTENANCE	:=1,	(* Maintenance hint *)
																			TCEVENTCLASS_MESSAGE		:=2,	(* Message *)
																			TCEVENTCLASS_HINT			:=3,	(* Hint *)
																			TCEVENTCLASS_STATEINFO		:=4,	(* State information *)
																			TCEVENTCLASS_INSTRUCTION	:=5,	(* Instruction *)
																			TCEVENTCLASS_WARNING		:=6,	(* Warning *)
																			TCEVENTCLASS_ALARM			:=7,	(* Alarm *)
																			TCEVENTCLASS_PARAMERROR		:=8		(* Parameter error *)  *)
	NoOfActiveEvents										:	INT;
END_VAR                                                 	
VAR                                                     	
	_Mem													:	BYTE;
	Disabled												:	BOOL;
	i 														:	INT;
END_VAR

(* EventHandlingGrp			V4.1	*)
(************************************)

(* status ***************************)
Status  													:= 0;
NoOfActiveEvents											:= 0;

IF(Disable OR SourceId = 0)AND Disabled
THEN
	RETURN;
ELSE
	Disabled												:= Disable OR SourceId = 0;
	
	FOR i := MIN_EVENT TO MAX_EVENT 
	DO
		(* Init Default Class *)
		IF SetClass <> TC2_SYSTEM.TCEVENTCLASS_ALARM
			AND NOT _Mem.7
		THEN
			no[i].eClass										:= SetClass;
			_Mem.7											:= i = MAX_EVENT;
		END_IF                                  			
		                                        			
		IF Disable OR SourceId = 0              			
		THEN                                    			
			no[i].Flag 										:= FALSE;
			no[i].ConfirmTrig 										:= no[i].State <> TCEVENTSTATE_INVALID AND no[i].State <> TCEVENTSTATE_RESETCON;
		ELSIF ConfirmTrig                             			
		THEN                                    	
			no[i].ConfirmTrig 								:= TRUE;
			_Mem.0 											:= ConfirmTrig;
                                                			
		ELSIF _Mem.0                            			
		THEN                                    			
			no[i].ConfirmTrig 								:= FALSE;
			_Mem.0 											:= i <> MAX_EVENT;

		ELSIF AutoConfirm
		THEN
			IF NOT no[i].Flag
				AND no[i].State <> TCEVENTSTATE_INVALID
				AND no[i].State <> TCEVENTSTATE_RESETCON
			THEN
				no[i].ConfirmTrig 							:= TRUE;
			ELSE                                			
				no[i].ConfirmTrig 							:= FALSE;
			END_IF                              			
		END_IF                                  	
                                                	
		(* Mem current Event *)                 	
		IF no[i].State <> TCEVENTSTATE_INVALID OR no[i].Flag 
		THEN
			_Mem.1											:= TRUE;
			(* Call Event *)
			no[i](
				Flag	:= ,
				ConfirmTrig := ,
				MsgId	:= TO_UINT(i + MsgOffset),
				SourceId:= SourceId,
				eClass	:= (* see grp call *),
				Text1	:= (* see grp call *),
				Text2	:= (* see grp call *),
				pText3	:= (* see grp call *),
				State	=> );
		END_IF

		(* Set info flags *)
		IF	no[i].State <> TCEVENTSTATE_INVALID 
		THEN
			NoOfActiveEvents								:= NoOfActiveEvents + 1;
			Status											:= Status OR no[i].Status;
			Disabled										:= FALSE;
		ELSIF _Mem.1
		THEN (* Send one time info event is gone *)
			; 
		END_IF
	END_FOR	
END_IF
(*****************************************************************************************)

METHOD PUBLIC confirm : booL  //Return value = TRUE if execution finished
VAR_INPUT
END_VAR
IF NoOfActiveEvents > 0
THEN
	FOR i := MIN_EVENT TO MAX_EVENT 
	DO
		no[i](ConfirmTrig := TRUE);
	END_FOR
	_Mem.0			:= TRUE;
END_IF

confirm		:= TRUE;
END_METHOD

END_FUNCTION_BLOCK

// POUs/EventLogger/TriggerEvents/EventHandlingStatisticInfo
{attribute 'no_check'}
//Collection with count and class types of active events 
FUNCTION_BLOCK EventHandlingStatisticInfo
VAR_OUTPUT CONSTANT
	MIN_CLASS												: 	UINT := TCEVENTCLASS_NONE;
	MAX_CLASS												: 	UINT := TCEVENTCLASS_PARAMERROR;
	MIN_PRIORITY											: 	INT := 0;
	MAX_PRIORITY											: 	INT := 7;
END_VAR
VAR_INPUT
	ClassInfo												:	ARRAY[MIN_CLASS..MAX_CLASS] OF INT; (* No of active messages in each class
																										TCEVENTCLASS_NONE			:=0
																										TCEVENTCLASS_MAINTENANCE	:=1	
																										TCEVENTCLASS_MESSAGE		:=2
																										TCEVENTCLASS_HINT			:=3	
																										TCEVENTCLASS_STATEINFO		:=4	
																										TCEVENTCLASS_INSTRUCTION	:=5	
																										TCEVENTCLASS_WARNING		:=6	
																										TCEVENTCLASS_ALARM			:=7	
																										TCEVENTCLASS_PARAMERROR		:=8 *)
	PriorityInfo											:	ARRAY[MIN_PRIORITY..MAX_PRIORITY] OF INT; //No of active messages per priority - see Param.EVENT_HANDLING_CONFIG
	NoOfQuitRequiredEvents									:	INT;
	NoOfActiveEvents										:	INT;
END_VAR
VAR_OUTPUT
END_VAR
VAR
	TaskInterlockCountIn									:	BOOL;
	TaskInterlockCountOut									:	BOOL;
END_VAR

;

PROPERTY PUBLIC classAlarmActive : BOOL
GET
classAlarmActive													:= ClassInfo[TCEVENTCLASS_ALARM] <> 0;
END_GET
END_PROPERTY

PROPERTY PUBLIC classHintActive : BOOL
GET
classHintActive													:= ClassInfo[TCEVENTCLASS_HINT] <> 0;
END_GET
END_PROPERTY

PROPERTY PUBLIC classInstructionActive : BOOL
GET
classInstructionActive													:= ClassInfo[TCEVENTCLASS_INSTRUCTION] <> 0;
END_GET
END_PROPERTY

PROPERTY PUBLIC classMaintenanceActive : BOOL
GET
classMaintenanceActive													:= ClassInfo[TCEVENTCLASS_MAINTENANCE] <> 0;
END_GET
END_PROPERTY

PROPERTY PUBLIC classMessageActive : BOOL
GET
classMessageActive													:= ClassInfo[TCEVENTCLASS_MESSAGE] <> 0;
END_GET
END_PROPERTY

PROPERTY PUBLIC classNoneActive : BOOL
GET
ClassNoneActive													:= ClassInfo[TCEVENTCLASS_NONE] <> 0;
END_GET
END_PROPERTY

PROPERTY PUBLIC classParamErrorActive : BOOL
GET
ClassParamErrorActive													:= ClassInfo[TCEVENTCLASS_PARAMERROR] <> 0;
END_GET
END_PROPERTY

PROPERTY PUBLIC classStateinfoActive : BOOL
GET
ClassStateinfoActive													:= ClassInfo[TCEVENTCLASS_STATEINFO] <> 0;
END_GET
END_PROPERTY

PROPERTY PUBLIC classWarningActive : BOOL
GET
ClassWarningActive													:= ClassInfo[TCEVENTCLASS_WARNING] <> 0;
END_GET
END_PROPERTY

METHOD PUBLIC clear : BOOL //Return value = TRUE if execution finished 
VAR_INPUT
END_VAR
	MEMSET(ADR(ClassInfo),0,SIZEOF(ClassInfo));
	MEMSET(ADR(PriorityInfo),0,SIZEOF(PriorityInfo));
	NoOfQuitRequiredEvents									:= 0;	
	NoOfActiveEvents										:= 0;
	Clear													:= TRUE;
END_METHOD

{attribute 'hide'}
METHOD PUBLIC countIn : BOOL //Return value = TRUE if execution finished 
VAR_IN_OUT
	Status													:	DWORD; (*	.0 - .8 = event of <class id> is active / .15 confirm required / .16 = Level 0 , .17 = Level 1 , .18 = Level 2, ..........
																			TCEVENTCLASS_NONE			:=0,	(* No class *)
																			TCEVENTCLASS_MAINTENANCE	:=1,	(* Maintenance hint *)
																			TCEVENTCLASS_MESSAGE		:=2,	(* Message *)
																			TCEVENTCLASS_HINT			:=3,	(* Hint *)
																			TCEVENTCLASS_STATEINFO		:=4,	(* State information *)
																			TCEVENTCLASS_INSTRUCTION	:=5,	(* Instruction *)
																			TCEVENTCLASS_WARNING		:=6,	(* Warning *)
																			TCEVENTCLASS_ALARM			:=7,	(* Alarm *)
																			TCEVENTCLASS_PARAMERROR		:=8		(* Parameter error *)  *)
END_VAR
IF TestAndSet(TaskInterlockCountIn)
THEN
	IF Status.0 THEN ClassInfo[TCEVENTCLASS_NONE] 				:= ClassInfo[TCEVENTCLASS_NONE] + 1; 									
	ELSIF Status.1 THEN ClassInfo[TCEVENTCLASS_MAINTENANCE] 	:= ClassInfo[TCEVENTCLASS_MAINTENANCE] + 1; 
	ELSIF Status.2 THEN ClassInfo[TCEVENTCLASS_MESSAGE] 		:= ClassInfo[TCEVENTCLASS_MESSAGE] + 1; 	
	ELSIF Status.3 THEN ClassInfo[TCEVENTCLASS_HINT] 			:= ClassInfo[TCEVENTCLASS_HINT] + 1; 		
	ELSIF Status.4 THEN ClassInfo[TCEVENTCLASS_STATEINFO] 		:= ClassInfo[TCEVENTCLASS_STATEINFO] + 1; 	
	ELSIF Status.5 THEN ClassInfo[TCEVENTCLASS_INSTRUCTION] 	:= ClassInfo[TCEVENTCLASS_INSTRUCTION] + 1; 
	ELSIF Status.6 THEN ClassInfo[TCEVENTCLASS_WARNING] 		:= ClassInfo[TCEVENTCLASS_WARNING] + 1; 	
	ELSIF Status.7 THEN ClassInfo[TCEVENTCLASS_ALARM] 			:= ClassInfo[TCEVENTCLASS_ALARM] + 1; 		
	ELSIF Status.8 THEN ClassInfo[TCEVENTCLASS_PARAMERROR] 		:= ClassInfo[TCEVENTCLASS_PARAMERROR] + 1; 	
	END_IF
	
	IF Status.15 THEN NoOfQuitRequiredEvents 					:= NoOfQuitRequiredEvents + 1; END_IF
	
	IF status.16 THEN PriorityInfo[0]							:= PriorityInfo[0] + 1;						
	ELSIF status.17 THEN PriorityInfo[1]						:= PriorityInfo[1] + 1	;						
	ELSIF status.18 THEN PriorityInfo[2]						:= PriorityInfo[2] + 1;						
	ELSIF status.19 THEN PriorityInfo[3]						:= PriorityInfo[3] + 1;						
	ELSIF status.20 THEN PriorityInfo[4]						:= PriorityInfo[4] + 1;						
	ELSIF status.21 THEN PriorityInfo[5]						:= PriorityInfo[5] + 1;						
	ELSIF status.22 THEN PriorityInfo[6]						:= PriorityInfo[6] + 1;						
	ELSIF status.23 THEN PriorityInfo[7]						:= PriorityInfo[7] + 1	;						
	END_IF
	
	//set active flag	
	NoOfActiveEvents											:= NoOfActiveEvents + 1;
	
	status.31 													:= TRUE; 
	CountIn														:= TRUE;
	TaskInterlockCountIn										:= FALSE;
END_IF
END_METHOD

// {attribute 'hide'}
METHOD PUBLIC countOut : BOOL //Return value = TRUE if execution finished 
VAR_IN_OUT
	Status													:	DWORD; (*	.0 - .8 = event of <class id> is active / .15 confirm required / .16 = Level 0 , .17 = Level 1 , .18 = Level 2, ..........
																			TCEVENTCLASS_NONE			:=0,	(* No class *)
																			TCEVENTCLASS_MAINTENANCE	:=1,	(* Maintenance hint *)
																			TCEVENTCLASS_MESSAGE		:=2,	(* Message *)
																			TCEVENTCLASS_HINT			:=3,	(* Hint *)
																			TCEVENTCLASS_STATEINFO		:=4,	(* State information *)
																			TCEVENTCLASS_INSTRUCTION	:=5,	(* Instruction *)
																			TCEVENTCLASS_WARNING		:=6,	(* Warning *)
																			TCEVENTCLASS_ALARM			:=7,	(* Alarm *)
																			TCEVENTCLASS_PARAMERROR		:=8		(* Parameter error *)  *)
END_VAR
IF TestAndSet(TaskInterlockCountOut)
THEN
	IF Status.0 THEN ClassInfo[TCEVENTCLASS_NONE] 				:= MAX(0,ClassInfo[TCEVENTCLASS_NONE] - 1); 		
	ELSIF Status.1 THEN ClassInfo[TCEVENTCLASS_MAINTENANCE] 	:= MAX(0,ClassInfo[TCEVENTCLASS_MAINTENANCE] - 1);	
	ELSIF Status.2 THEN ClassInfo[TCEVENTCLASS_MESSAGE] 		:= MAX(0,ClassInfo[TCEVENTCLASS_MESSAGE] - 1); 		
	ELSIF Status.3 THEN ClassInfo[TCEVENTCLASS_HINT] 			:= MAX(0,ClassInfo[TCEVENTCLASS_HINT] - 1); 		
	ELSIF Status.4 THEN ClassInfo[TCEVENTCLASS_STATEINFO] 		:= MAX(0,ClassInfo[TCEVENTCLASS_STATEINFO] - 1); 	
	ELSIF Status.5 THEN ClassInfo[TCEVENTCLASS_INSTRUCTION] 	:= MAX(0,ClassInfo[TCEVENTCLASS_INSTRUCTION] - 1);	
	ELSIF Status.6 THEN ClassInfo[TCEVENTCLASS_WARNING] 		:= MAX(0,ClassInfo[TCEVENTCLASS_WARNING] - 1); 	
	ELSIF Status.7 THEN ClassInfo[TCEVENTCLASS_ALARM] 			:= MAX(0,ClassInfo[TCEVENTCLASS_ALARM] - 1); 		
	ELSIF Status.8 THEN ClassInfo[TCEVENTCLASS_PARAMERROR] 		:= MAX(0,ClassInfo[TCEVENTCLASS_PARAMERROR] - 1); 	
	END_IF
																	  
	IF Status.15 THEN NoOfQuitRequiredEvents 					:=  MAX(0,NoOfQuitRequiredEvents - 1); 	
	END_IF
																	   
	IF status.16 THEN PriorityInfo[0]							:=  MAX(0,PriorityInfo[0] - 1);						
	ELSIF status.17 THEN PriorityInfo[1]						:=  MAX(0,PriorityInfo[1] - 1);						
	ELSIF status.18 THEN PriorityInfo[2]						:=  MAX(0,PriorityInfo[2] - 1);						
	ELSIF status.19 THEN PriorityInfo[3]						:=  MAX(0,PriorityInfo[3] - 1);						
	ELSIF status.20 THEN PriorityInfo[4]						:=  MAX(0,PriorityInfo[4] - 1);						
	ELSIF status.21 THEN PriorityInfo[5]						:=  MAX(0,PriorityInfo[5] - 1);						
	ELSIF status.22 THEN PriorityInfo[6]						:=  MAX(0,PriorityInfo[6] - 1);						
	ELSIF status.23 THEN PriorityInfo[7]						:=  MAX(0,PriorityInfo[7] - 1);						
	END_IF
	
	NoOfActiveEvents											:= MAX(0,NoOfActiveEvents - 1);
	status.31													:= FALSE; //Active flag reset
	CountOut													:= TRUE;
	TaskInterlockCountOut										:= FALSE;
END_IF
END_METHOD

METHOD INTERNAL initEvent : DWORD //Return status 
VAR_IN_OUT
	SetClass								:	E_TcEventClass;
	EventConfig								:	TcEvent;
END_VAR
		(* Event Config *)
		InitEvent											:= 0;
		IF SetClass = TC2_SYSTEM.TCEVENTCLASS_NONE 				
		THEN	
			EventConfig.Class								:= SetClass;
			EventConfig.bQuitRequired						:= PARAM.EVENT_HANDLING_CONFIG.CLASS_NONE_QUIT_REQUIRED;
			InitEvent.15									:= PARAM.EVENT_HANDLING_CONFIG.CLASS_NONE_QUIT_REQUIRED;
			EventConfig.Prio								:= PARAM.EVENT_HANDLING_CONFIG.CLASS_NONE_PRIORITY;
			InitEvent										:= SETBIT32(InitEvent,TO_SINT(PARAM.EVENT_HANDLING_CONFIG.CLASS_NONE_PRIORITY) + 16);	
			InitEvent.0										:= TRUE;													
			
		ELSIF SetClass = TC2_SYSTEM.TCEVENTCLASS_MAINTENANCE 
		THEN
			EventConfig.Class								:= SetClass;
			EventConfig.bQuitRequired						:= PARAM.EVENT_HANDLING_CONFIG.CLASS_MAINTENANCE_QUIT_REQUIRED;
			InitEvent.15									:= PARAM.EVENT_HANDLING_CONFIG.CLASS_MAINTENANCE_QUIT_REQUIRED;
			EventConfig.Prio								:= PARAM.EVENT_HANDLING_CONFIG.CLASS_MAINTENANCE_PRIORITY;
			InitEvent										:= SETBIT32(InitEvent,TO_SINT(PARAM.EVENT_HANDLING_CONFIG.CLASS_MAINTENANCE_PRIORITY) + 16);
			InitEvent.1										:= TRUE;
		ELSIF SetClass = TC2_SYSTEM.TCEVENTCLASS_MESSAGE 		
		THEN
			EventConfig.Class								:= SetClass;
			EventConfig.bQuitRequired						:= PARAM.EVENT_HANDLING_CONFIG.CLASS_MESSAGE_QUIT_REQUIRED;
			InitEvent.15									:= PARAM.EVENT_HANDLING_CONFIG.CLASS_MESSAGE_QUIT_REQUIRED;
			EventConfig.Prio								:= PARAM.EVENT_HANDLING_CONFIG.CLASS_MESSAGE_PRIORITY;
			InitEvent										:= SETBIT32(InitEvent,TO_SINT(PARAM.EVENT_HANDLING_CONFIG.CLASS_MESSAGE_PRIORITY) + 16);
			InitEvent.2										:= TRUE;
		ELSIF SetClass = TC2_SYSTEM.TCEVENTCLASS_HINT 			
		THEN
			EventConfig.Class								:= SetClass;
			EventConfig.bQuitRequired						:= PARAM.EVENT_HANDLING_CONFIG.CLASS_HINT_QUIT_REQUIRED;
			InitEvent.15									:= PARAM.EVENT_HANDLING_CONFIG.CLASS_HINT_QUIT_REQUIRED;
			EventConfig.Prio								:= PARAM.EVENT_HANDLING_CONFIG.CLASS_HINT_PRIORITY;
			InitEvent										:= SETBIT32(InitEvent,TO_SINT(PARAM.EVENT_HANDLING_CONFIG.CLASS_HINT_PRIORITY) + 16);
			InitEvent.3										:= TRUE;
		ELSIF SetClass = TC2_SYSTEM.TCEVENTCLASS_STATEINFO 	
		THEN
			EventConfig.Class								:= SetClass;
			EventConfig.bQuitRequired						:= PARAM.EVENT_HANDLING_CONFIG.CLASS_STATEINFO_QUIT_REQUIRED;
			InitEvent.15									:= PARAM.EVENT_HANDLING_CONFIG.CLASS_STATEINFO_QUIT_REQUIRED;
			EventConfig.Prio								:= PARAM.EVENT_HANDLING_CONFIG.CLASS_STATEINFO_PRIORITY;
			InitEvent										:= SETBIT32(InitEvent,TO_SINT(PARAM.EVENT_HANDLING_CONFIG.CLASS_STATEINFO_PRIORITY) + 16);
			InitEvent.4										:= TRUE;
		ELSIF SetClass = TC2_SYSTEM.TCEVENTCLASS_INSTRUCTION 
		THEN
			EventConfig.Class								:= SetClass;
			EventConfig.bQuitRequired						:= PARAM.EVENT_HANDLING_CONFIG.CLASS_INSTRUCTION_QUIT_REQUIRED;
			InitEvent.15									:= PARAM.EVENT_HANDLING_CONFIG.CLASS_INSTRUCTION_QUIT_REQUIRED;
			EventConfig.Prio								:= PARAM.EVENT_HANDLING_CONFIG.CLASS_INSTRUCTION_PRIORITY;
			InitEvent										:= SETBIT32(InitEvent,TO_SINT(PARAM.EVENT_HANDLING_CONFIG.CLASS_INSTRUCTION_PRIORITY) + 16);
			InitEvent.5										:= TRUE;
		ELSIF SetClass = TC2_SYSTEM.TCEVENTCLASS_WARNING 		
		THEN
			EventConfig.Class								:= SetClass;
			EventConfig.bQuitRequired						:= PARAM.EVENT_HANDLING_CONFIG.CLASS_WARNING_QUIT_REQUIRED;
			InitEvent.15									:= PARAM.EVENT_HANDLING_CONFIG.CLASS_WARNING_QUIT_REQUIRED;
			EventConfig.Prio								:= PARAM.EVENT_HANDLING_CONFIG.CLASS_WARNING_PRIORITY;
			InitEvent										:= SETBIT32(InitEvent,TO_SINT(PARAM.EVENT_HANDLING_CONFIG.CLASS_WARNING_PRIORITY) + 16);
			InitEvent.6										:= TRUE;
		ELSIF SetClass = TC2_SYSTEM.TCEVENTCLASS_ALARM 		
		THEN
			EventConfig.Class								:= SetClass;
			EventConfig.bQuitRequired						:= PARAM.EVENT_HANDLING_CONFIG.CLASS_ALARM_QUIT_REQUIRED;
			InitEvent.15									:= PARAM.EVENT_HANDLING_CONFIG.CLASS_ALARM_QUIT_REQUIRED;
			EventConfig.Prio								:= PARAM.EVENT_HANDLING_CONFIG.CLASS_ALARM_PRIORITY;
			InitEvent										:= SETBIT32(InitEvent,TO_SINT(PARAM.EVENT_HANDLING_CONFIG.CLASS_ALARM_PRIORITY) + 16);
			InitEvent.7										:= TRUE;
		ELSIF SetClass = TC2_SYSTEM.TCEVENTCLASS_PARAMERROR 	
		THEN
			EventConfig.Class								:= SetClass;
			EventConfig.bQuitRequired						:= PARAM.EVENT_HANDLING_CONFIG.CLASS_PARAMERROR_QUIT_REQUIRED;
			InitEvent.15									:= PARAM.EVENT_HANDLING_CONFIG.CLASS_PARAMERROR_QUIT_REQUIRED;
			EventConfig.Prio								:= PARAM.EVENT_HANDLING_CONFIG.CLASS_PARAMERROR_PRIORITY;
			InitEvent										:= SETBIT32(InitEvent,TO_SINT(PARAM.EVENT_HANDLING_CONFIG.CLASS_PARAMERROR_PRIORITY) + 16);
			InitEvent.8										:= TRUE;
		ELSE 
			EventConfig.Class								:= SetClass;
			EventConfig.bQuitRequired						:= PARAM.EVENT_HANDLING_CONFIG.CLASS_ALARM_QUIT_REQUIRED;
			InitEvent.15									:= PARAM.EVENT_HANDLING_CONFIG.CLASS_ALARM_QUIT_REQUIRED;
			EventConfig.Prio								:= PARAM.EVENT_HANDLING_CONFIG.CLASS_ALARM_PRIORITY;
			InitEvent										:= SETBIT32(InitEvent,TO_SINT(PARAM.EVENT_HANDLING_CONFIG.CLASS_ALARM_PRIORITY) + 16);
			InitEvent.7										:= TRUE;
		END_IF
END_METHOD

METHOD PUBLIC isClassActive : BOOL  //Return value = TRUE if EventClass is currently active
VAR_INPUT
	TcEventClass											:	E_TcEventClass;
END_VAR
IF TcEventClass < MIN_CLASS OR TcEventClass > MAX_CLASS
THEN
	IsClassActive											:= TRUE;
ELSE
	IsClassActive											:= ClassInfo[TcEventClass] <> 0;
END_IF
END_METHOD

PROPERTY PUBLIC isConfirmReqActive : BOOL
GET
isConfirmReqActive											:= NoOfQuitRequiredEvents <> 0;
END_GET
END_PROPERTY

METHOD PUBLIC isPriorityActive : BOOL //Return value = TRUE if priority is active
VAR_INPUT
	IN														:	INT;
END_VAR
IF IN < MIN_PRIORITY OR IN > MAX_PRIORITY
THEN
	IsPriorityActive										:= TRUE;
ELSE
	IsPriorityActive										:= PriorityInfo[In] <> 0;
END_IF
END_METHOD

END_FUNCTION_BLOCK

// POUs/EventLogger/EventsWriteToLogbook
{attribute 'no_check'}
//Write new event logger messages from "ReadAdsEvent" instance into "LogBook" instance
FUNCTION_BLOCK EventsWriteToLogbook
VAR_OUTPUT CONSTANT
{attribute 'displaymode':='binary'}
	OPTION_ADD_DT_TO_MSG_STRING								:	BYTE := 2#0000_0001;
{attribute 'displaymode':='binary'}
	OPTION_ADD_CLASS_TO_MSG_STRING							:	BYTE := 2#0000_0010;
{attribute 'displaymode':='binary'}
	OPTION_ADD_SOURCE_TO_MSG_STRING							:	BYTE := 2#0000_0100;	//Default option
{attribute 'displaymode':='binary'}
	OPTION_ADD_SOURCE_ID_TO_MSG_STRING						:	BYTE := 2#0000_1000; 
{attribute 'displaymode':='binary'}
	OPTION_ADD_MSG_ID_TO_MSG_STRING							:	BYTE := 2#0001_0000;	//Default option	
{attribute 'displaymode':='binary'}
	OPTION_ADD_MSG_DT_TO_LOGBOOK_TIMESTAMP					:	BYTE := 2#0010_0000;	
{attribute 'displaymode':='binary'}
	OPTION_ADD_MSG_STATE_ID_TO_MSG_STRING					:	BYTE := 2#0100_0000;	//Add event state before text
END_VAR
VAR_INPUT
	Enable													:	BOOL	:= FALSE;	//Activate the function block
{attribute 'displaymode':='binary'}
	Options													:	BYTE 	:= OPTION_ADD_SOURCE_TO_MSG_STRING OR OPTION_ADD_MSG_ID_TO_MSG_STRING;
END_VAR                                                     
VAR_IN_OUT                                                  
	EventlogRead											:	EventlogRead;		//ReadAdsEvent instance
	LogBook													:	LogBook_wEventClass;//Logbook instance 
END_VAR                                                     
VAR_OUTPUT                                                  
	LastEventDT												:	DT;					//Date and time of last checked event
END_VAR                                                         			
VAR
(* Memory ******************************************************)
	LastEntryTimestamp										:	T_DCTIME64;			//Date of last event in this cycle
	LastEventTimestamp										:	T_DCTIME64;			//Timestamp of last added event
	ExitMarker												:	BOOL;
	MemLogbookOptions										:	BYTE;	
	MemClass												:	E_TcEventClass := TC2_SYSTEM.TCEVENTCLASS_ALARM;
	MemTimestamp											:	TIMESTRUCT;
	LenMem													:	INT;

	
(* Timer *******************************************************)

(* Trigger *****************************************************)

(* Blocks ******************************************************)

(* Error *******************************************************)

(* Dummys ******************************************************)
	i														: 	INT := 0; 
	k,j														:	INT;
	OK														:	BOOL;
END_VAR

(* Read new events and write into logbook 							*)
(********************************************************************)

(* action ***********************************************************)
IF Enable 
THEN
	IF EventlogRead.Done
	THEN //Start read events
	
		//first save Logbook settings 
		MemTimestamp										:= LogBook.Timestamp;
		MemLogbookOptions									:= LogBook.Options;		
		MemClass											:= LogBook.Class;
	(*	LogBook.Options										:= LogBook.Options 
																AND Logbook.OPTION_WRITE_TO_ADSLOG AND Logbook.OPTION_WRITE_TO_FILE 
																AND Logbook.OPTION_ADD_TIME_TO_MSG_STRING AND Logbook.OPTION_ADD_TIME_TO_MSG_STRING ; *)
		
		//Check list for new entrys
		ExitMarker											:= FALSE;
		FOR i := EventlogRead.TotalNumberOfEvents TO EventlogRead.MIN_EVENT BY - 1  
		DO
			IF EventlogRead.Event[i].Timestamp > LastEntryTimestamp
			THEN //New entries
				IF NOT ExitMarker 
					OR //Events with event newer timestamp, exit and continue at next cycle
					EventlogRead.Event[i].Timestamp = LastEventTimestamp
				THEN //new message
					ExitMarker								:= TRUE;
					LastEventTimestamp						:= EventlogRead.Event[i].Timestamp;
										
					IF _formatMsg(EventlogRead.LangId, EventlogRead.Event[i], LogBook)
					THEN //Write message to logbook	
						Logbook();
					END_IF
					
				ELSE //add messages the next time
					EXIT; 
				END_IF
				
			ELSE //old messages
				;
			END_IF
		
		END_FOR		
		
		//Record timestamp of last event
		LastEntryTimestamp									:= LastEventTimestamp;

		//Recover old entries	
		LogBook.Options										:= MemLogbookOptions;
		LogBook.Class										:= MemClass;
		LogBook.Timestamp									:= MemTimestamp;				
	END_IF	
END_IF

(*******************************************************************************)

METHOD PROTECTED _formatMsg : BOOL
VAR_INPUT
	Lcid													:	eLCID;
END_VAR
VAR_IN_OUT
	Event													 : EVENTLOG_READ_DATA;
	LogBook													:	LogBook_wEventClass;//Logbook instance 
END_VAR
//2020-05-30-07:06:08.436;<EventClass txt>;<Source ID>;<Event Id>;<Event state>;CoE Drive | AxisY - Remote control over fieldbus not active  	

	//Add class to log book entry
	LogBook.Class											:= Event.Class;	
	Logbook.Msg												:= '';
	
	//Event timestamp to logbook timestamp
	IF OPtions.5
	THEN
		LogBook.Timestamp 									:= DT_TO_SYSTEMTIME(Event.TimestampDT);			
	END_IF
	
	//add date and time
	IF Options.0
	THEN					
		LogBook.Msg											:= DT_TO_STRING(Event.TimestampDT);			
		LogBook.Msg											:= DELETE(LogBook.Msg, 3, 1); //delete DT# 
		LogBook.Msg 										:= CONCAT(LogBook.Msg,';');					
	END_IF
		
	//add event class
	IF Options.1
	THEN
		LogBook.Msg											:= CONCAT(LogBook.Msg,GetEventClassText(Event.Class));
		LogBook.Msg 										:= CONCAT(LogBook.Msg,';');
	END_IF

	//add source id 
	IF Options.3 
	THEN
		LogBook.Msg 										:= CONCAT(LogBook.Msg,TO_STRING(Event.Sourceid));
		LogBook.Msg 										:= CONCAT(LogBook.Msg,';');		
	END_IF							
							
	//add event id 
	IF Options.4
	THEN
		LogBook.Msg 										:= CONCAT(LogBook.Msg,DWORD_TO_STRING(Event.id));
		LogBook.Msg 										:= CONCAT(LogBook.Msg,';');				
	END_IF					
	
	//add event state
	IF Options.6
	THEN
		LogBook.Msg 										:= CONCAT(LogBook.Msg,DWORD_TO_STRING(Event.State));
		LogBook.Msg 										:= CONCAT(LogBook.Msg,';');				
	END_IF					

	//add event source text
	IF Options.2
	THEN
		IF Lcid <> eLCID.CN
		THEN
			LogBook.Msg 									:= CONCAT(LogBook.Msg,WSTRING_TO_STRING(Event.Source));
			LogBook.Msg 									:= CONCAT(LogBook.Msg,' | ');	
		ELSIF NOT Options.3    
		THEN                               
			LogBook.Msg 									:= CONCAT(LogBook.Msg,CONCAT('Source Id[', UDINT_TO_STRING(Event.Sourceid)));
			LogBook.Msg 									:= CONCAT(LogBook.Msg,'] | ');								
		END_IF	
	END_IF
		
	IF Lcid <> eLCID.CN
	THEN
		LogBook.Msg											:= CONCAT(LogBook.Msg,WSTRING_TO_STRING(Event.MsgText));
	ELSE
		LogBook.Msg 										:= CONCAT(LogBook.Msg, SEL(Options.4 , CONCAT('EventId[' ,CONCAT(UDINT_TO_STRING(Event.id),'] <Unicode active>')) , '<Unicode active>'));										
	END_IF

	_formatMsg												:= TRUE;
	
(**********************************************************************************************)
END_METHOD

END_FUNCTION_BLOCK

// POUs/Logging/Logbook
{attribute 'no_check'}
//PLC Logbook for debugging, records a number of "MAX_DATA" messages with timestamp.
//The Logbook Puplisher can be used to forward messages from the logbook to several subscriber (Write into Logfile, display via EventLogger, send to Syslog Server)
//
//Parameter Timestamp needs to be updated externaly every cycle if needed
//
//Function "LogWithEventClass" is used inside
FUNCTION_BLOCK Logbook IMPLEMENTS I_Logbook                 									
VAR_OUTPUT CONSTANT     									
//Parameter
	MIN_DATA												:	INT := 1;
	MAX_DATA												:	INT := PARAM.LOGBOOK_MAX_DATA; //see library parameter to customize parameter	
                        									
//option settings to modify the message string and behavior
{attribute 'displaymode':='binary'}
	OPTION_WRITE_TO_ADSLOG									: 	BYTE :=2#0000_0100; //Write entry directly to TwinCAT logger (shown in XAE output)
{attribute 'displaymode':='binary'}
	OPTION_ADD_TIME_TO_MSG_STRING							: 	BYTE :=2#0000_1000;	//Add time stamp to message string 
{attribute 'displaymode':='binary'}
	OPTION_ADD_DATE_TO_MSG_STRING							: 	BYTE :=2#0001_0000; //Add date to message string
END_VAR                 									
VAR_INPUT               									                       		
{attribute 'displaymode':='binary'}
	Options													:	BYTE := 2#0000_0000;			(* option constants are alreay predefined, so they can accordingly be passed symbolically to the block
																								Bit 0 = 
																								Bit 1 = 
																								Bit 2 = Send to TC Ads-Logger
																								Bit 3 = Add time to message string
																								Bit 4 = Add date to message string
																								Bit 5 = 
																								Bit 6 = 
														 										Bit 7 =  								
																								*)
                        									
// InputData         	
	Timestamp												:	TIMESTRUCT; //Time stamp need to be updated cylic if it will be used
	Msg														:	STRING(PARAM.LOGBOOK_MAX_MSG_STRING_LENGHT) := ''; //Message string which will written into the DataMsg array by executing the Fb																							
END_VAR             										
VAR_OUTPUT
	Data													:	ARRAY[MIN_DATA..MAX_DATA] OF LogbookData; // Recorded messages data
	CntAddedMessages										:	INT;
END_VAR
VAR
	TaskInterlock											:	BOOL;
END_VAR

(* LogBook 									 *)
(*********************************************)

(* call method *********************************************)
	_Write(Msg);
(***********************************************************)

METHOD PROTECTED _write : BOOL
VAR_IN_OUT
	Msg														:	STRING(PARAM.LOGBOOK_MAX_MSG_STRING_LENGHT);
END_VAR
(* Write entry with every call ******************************)
IF LEN(MSG) = 0
THEN
	_Write													:= FALSE;
	RETURN;
ELSIF TestAndSet(TaskInterlock)
THEN	
	MEMMOVE(ADR(Data[MIN(MIN_DATA + 1,MAX_DATA)]), 	ADR(Data), 	SIZEOF(Data) - SIZEOF(Data[MIN_DATA]));
	
	(* Datensatz oben eintragen *)
	IF NOT Options.3 AND NOT Options.4
	THEN
		Data[MIN_DATA].Msg									:= Msg;
	ELSIF Options.3 AND Options.4              
	THEN                                                    
		Data[MIN_DATA].Msg									:= SYSTEMTIME_TO_STRING(Timestamp);
		Data[MIN_DATA].Msg									:= CONCAT(Data[MIN_DATA].Msg, ' | ');
		Data[MIN_DATA].Msg									:= CONCAT(Data[MIN_DATA].Msg, Msg);
	ELSIF Options.4                                   
	THEN                                                    
		Data[MIN_DATA].Msg									:= SYSTEMTIME_TO_STRING(Timestamp);
		Data[MIN_DATA].Msg									:=	MID(Data[MIN_DATA].Msg, 12 , 12);
		Data[MIN_DATA].Msg									:= CONCAT(Data[MIN_DATA].Msg, ' | ');
		Data[MIN_DATA].Msg									:= CONCAT(Data[MIN_DATA].Msg, Msg);
                                                            
	ELSE (* Only Date to Msg String *)                      
		Data[MIN_DATA].Msg									:= SYSTEMTIME_TO_STRING(Timestamp);
		Data[MIN_DATA].Msg									:= MID(Data[MIN_DATA].Msg, 8 , 3);
		Data[MIN_DATA].Msg									:= CONCAT(Data[MIN_DATA].Msg, ' | ');
		Data[MIN_DATA].Msg									:= CONCAT(Data[MIN_DATA].Msg, Msg);
	END_IF                                                  

	//Coyp current options from logbook into message	                                                        
	Data[MIN_DATA].Options									:= TO_WORD(Options);
		
	//Store time stamp
	Data[MIN_DATA].Timestamp								:= Timestamp;
	
	CntAddedMessages										:= MIN(MAX_DATA, CntAddedMessages + 1); 
	_Write													:= TRUE;
	TaskInterlock											:= FALSE;
END_IF

(************************************************************)
END_METHOD

METHOD PUBLIC delete : BOOL //Return value = TRUE if execution finished
VAR_INPUT
END_VAR

CntAddedMessages											:= 0;
MEMSET(ADR(Data),0,SIZEOF(Data));
delete														:= TRUE;
END_METHOD

METHOD PUBLIC getOldestMsg : BOOL //Return value TRUE = if finished successful -> new message read
VAR_IN_OUT
	data													: LogbookData;								
END_VAR
IF CntAddedMessages >= MIN_DATA AND CntAddedMessages <= MAX_DATA
	AND NOT TaskInterlock
THEN
	data													:= THIS^.Data[CntAddedMessages];
	THIS^.Data[CntAddedMessages].Options.15					:= FALSE; //New message
	CntAddedMessages										:= CntAddedMessages - 1;
	getOldestMsg											:= TRUE;
ELSE
	getOldestMsg											:= FALSE;
END_IF
END_METHOD

PROPERTY PUBLIC optAddDateToMsgText : BOOL
GET
optAddDateToMsgText := Options.4;
END_GET
SET
Options.4 := optAddDateToMsgText;
END_SET
END_PROPERTY

PROPERTY PUBLIC optAddTimeToMsgText : BOOL
GET
optAddTimeToMsgText := Options.3;
END_GET
SET
Options.3 := optAddTimeToMsgText;
END_SET
END_PROPERTY

PROPERTY Public optWiteEntryToTcAdsLogger : BOOL
GET
optWiteEntryToTcAdsLogger := Options.2;
END_GET
SET
Options.2 := optWiteEntryToTcAdsLogger;
END_SET
END_PROPERTY

{attribute 'monitoring' := 'call'}
PROPERTY PUBLIC rCntAddedMessages : Reference to INT //Reference to variable showing no of added messages (Counter will be decreased by getOldestMsg)
GET
rCntAddedMessages REF= CntAddedMessages;
END_GET
END_PROPERTY

METHOD PUBLIC readMsg : REFERENCE TO LogbookData //Return value is a REFERENCE to the by Index selected entry.  
VAR_INPUT
	Index											:	INT;						
END_VAR

readMsg													REF= THIS^.Data[LIMIT(MIN_DATA,Index,MAX_DATA)];
END_METHOD

METHOD PUBLIC write : BOOL //Return value = TRUE if execution finished
VAR_INPUT
	Msg														:	STRING(PARAM.LOGBOOK_MAX_MSG_STRING_LENGHT);
END_VAR

write														:= _Write(Msg);
IF options.2 
THEN
	write 													:= write AND 0 = adsLogHint(Msg, '');
END_IF
END_METHOD

END_FUNCTION_BLOCK

// POUs/Logging/I_Logbook
INTERFACE I_Logbook Extends __System.IQueryInterface

METHOD PUBLIC delete : BOOL //Return value = TRUE if execution finished
VAR_INPUT
END_VAR
END_METHOD

METHOD PUBLIC getOldestMsg : BOOL //Return value TRUE = if finished successful -> new message flag of entry will be reset
VAR_IN_OUT
	data													: LogbookData;								
END_VAR
END_METHOD

{attribute 'monitoring' := 'call'}
PROPERTY PUBLIC rCntAddedMessages : Reference to INT
GET
END_GET
END_PROPERTY

METHOD PUBLIC readMsg : REFERENCE TO LogbookData //Return value is a REFERENCE to the by Index selected entry.  
VAR_INPUT
	Index											:	INT;						
END_VAR
END_METHOD

METHOD PUBLIC write : BOOL //Return value = TRUE if execution finished
VAR_INPUT
	Msg														:	STRING(PARAM.LOGBOOK_MAX_MSG_STRING_LENGHT);
END_VAR
END_METHOD

END_INTERFACE

// POUs/Logging/Logbook_wEventClass
{attribute 'no_check'}
FUNCTION_BLOCK Logbook_wEventClass EXTENDS Logbook             									
VAR_OUTPUT CONSTANT     									
END_VAR                 									
VAR_INPUT               									                       		
	Class													:	E_TcEventClass := TC2_SYSTEM.TCEVENTCLASS_NONE; //Possible event class for the entry																							
END_VAR             										
VAR_OUTPUT
END_VAR
VAR

END_VAR

(* LogBook 									 *)
(*********************************************)

(* call method *********************************************)
	Write(Msg);
(***********************************************************)

METHOD PUBLIC getClassFromOption : E_TcEventClass
VAR_INPUT
	Msgidx														:	INT;
END_VAR
IF Msgidx >= MIN_DATA AND Msgidx <= MAX_DATA
THEN
	GetClassFromOption.0 										:= Data[Msgidx].Options.8;
	GetClassFromOption.1 										:= Data[Msgidx].Options.9;
	GetClassFromOption.2 										:= Data[Msgidx].Options.10;
	GetClassFromOption.3 										:= Data[Msgidx].Options.11;
ELSE
	GetClassFromoption 											:= TCEVENTCLASS_ALARM;
END_IF
END_METHOD

METHOD PUBLIC write : BOOL //Return value = TRUE if execution finished
VAR_INPUT
	Msg														:	STRING(PARAM.LOGBOOK_MAX_MSG_STRING_LENGHT);
END_VAR

IF _Write(Msg)
THEN
	//Store class as integer in logbook options
	Data[MIN_DATA].Options.8								:= Class.0;
	Data[MIN_DATA].Options.9								:= Class.1; 
	Data[MIN_DATA].Options.10								:= Class.2; 
	Data[MIN_DATA].Options.11								:= Class.3;	
	write													:= TRUE;											
	
	IF options.2 
	THEN
		write												:= 0= adsLogwTcEventClass(Msg, Class);
	END_IF
END_IF
END_METHOD

METHOD PUBLIC writeWithClass : BOOL //Return value = TRUE if execution finished
VAR_INPUT
	Msg														:	STRING(PARAM.LOGBOOK_MAX_MSG_STRING_LENGHT);
	Class													:	E_TcEventClass := TC2_SYSTEM.TCEVENTCLASS_NONE;
END_VAR
IF _Write(Msg)
THEN
	//Store class as integer in logbook options
	Data[MIN_DATA].Options.8								:= Class.0;
	Data[MIN_DATA].Options.9								:= Class.1; 
	Data[MIN_DATA].Options.10								:= Class.2; 
	Data[MIN_DATA].Options.11								:= Class.3;	
	writeWithClass											:= TRUE;
	IF options.2 
	THEN
		writeWithClass 										:= 0 = adsLogwTcEventClass(Msg, Class);
	END_IF
END_IF
END_METHOD

END_FUNCTION_BLOCK

// POUs/Logging/adsLogwTcEventClass
{attribute 'no_check' := ''}
//Writing string as hint message into the TwinCAT ams logger and windows event log with a Lreal argument
//Please see Beckhoff information system "ADSLOGLREAL" for detailed information.
//Intention of this function is to use the handy ADSLOGxxxx without the annoying msgCtrlMask as a parameter :-)  
//Function "EventHandlingGetClassLevel" is used inside
FUNCTION adsLogwTcEventClass : DINT
VAR_INPUT               											
	MsgFmtStr												:	T_MaxString;
(*	dintArg													:	DINT; *) 
(*	strArg													:	T_MaxString; *)
(*	realArg													:	LREAL; *)
	TcEventClass											:	E_TcEventClass; 
END_VAR
VAR
	msgCtrlMask												:	DWORD; (* 	ADSLOG_MSGTYPE_HINT Meldungstyp ist Hinweis.
																				ADSLOG_MSGTYPE_WARN Meldungstyp ist Warnung.  
																				ADSLOG_MSGTYPE_ERROR Meldungstyp ist Fehler.  
																				ADSLOG_MSGTYPE_LOG Meldung wird in das Logbuch geschrieben.  
																				ADSLOG_MSGTYPE_MSGBOX Meldung wird in einer Messagebox ausgegeben.  
																				ADSLOG_MSGTYPE_RESOURCE Meldung wird aus einer Ressource-Datei geholt. (wird momentan nicht  unterstützt)  
																				ADSLOG_MSGTYPE_STRING 	Meldung ist direkt angegebener String (default).  *)	
END_VAR

(* create fixed message ctrl mask **********************************)
	CASE GetEventClassPriority(tcEventClass) OF 
	0:	msgCtrlMask											:= ADSLOG_MSGTYPE_HINT;
	1:	msgCtrlMask											:= ADSLOG_MSGTYPE_WARN;
	ELSE
		msgCtrlMask											:= ADSLOG_MSGTYPE_ERROR;
	END_CASE

	msgCtrlMask												:= ADSLOG_MSGTYPE_STRING OR msgCtrlMask OR ADSLOG_MSGTYPE_LOG;

(* write string which includes a floating-number ******************)
	adsLogwTcEventClass 										:= ADSLOGLREAL(msgCtrlMask, msgFmtStr, 0.0);
	
(* write string which includes a DINT-number *******************)
(*	LogWithEventClass 										:= ADSLOGDINT(msgCtrlMask, msgFmtStr, dintArg); *)

(* write string which includes an other string e.g. 'hallo: %s what's up' ***************)
(*	LogWithEventClass 										:= ADSLOGSTR(msgCtrlMask, msgFmtStr,msgCtrlMaskstrArg); *)

(*****************************************************)

END_FUNCTION

// POUs/EventLogger/getEventClassPriority
{attribute 'no_check'}
//Returns configured level to corresponding event class (see library Param) 
FUNCTION getEventClassPriority : UINT
VAR_INPUT
	TcEventClass											:	E_TcEventClass;
END_VAR
VAR
END_VAR

	CASE tcEventClass OF
	Tc2_System.TCEVENTCLASS_NONE:			GetEventClassPriority	:= PARAM.EVENT_HANDLING_CONFIG.CLASS_NONE_PRIORITY;	
	Tc2_System.TCEVENTCLASS_MAINTENANCE:	GetEventClassPriority	:= PARAM.EVENT_HANDLING_CONFIG.CLASS_MAINTENANCE_PRIORITY;		
	Tc2_System.TCEVENTCLASS_MESSAGE:		GetEventClassPriority	:= PARAM.EVENT_HANDLING_CONFIG.CLASS_MESSAGE_PRIORITY;			
	Tc2_System.TCEVENTCLASS_HINT:			GetEventClassPriority	:= PARAM.EVENT_HANDLING_CONFIG.CLASS_HINT_PRIORITY;	
	Tc2_System.TCEVENTCLASS_STATEINFO:		GetEventClassPriority	:= PARAM.EVENT_HANDLING_CONFIG.CLASS_STATEINFO_PRIORITY;	
	Tc2_System.TCEVENTCLASS_INSTRUCTION:	GetEventClassPriority	:= PARAM.EVENT_HANDLING_CONFIG.CLASS_INSTRUCTION_PRIORITY;	
	Tc2_System.TCEVENTCLASS_WARNING:		GetEventClassPriority	:= PARAM.EVENT_HANDLING_CONFIG.CLASS_WARNING_PRIORITY;	
	Tc2_System.TCEVENTCLASS_ALARM:			GetEventClassPriority	:= PARAM.EVENT_HANDLING_CONFIG.CLASS_ALARM_PRIORITY;	
	Tc2_System.TCEVENTCLASS_PARAMERROR:		GetEventClassPriority	:= PARAM.EVENT_HANDLING_CONFIG.CLASS_PARAMERROR_PRIORITY;		
	ELSE
		GetEventClassPriority										:= PARAM.EVENT_HANDLING_CONFIG.CLASS_ALARM_PRIORITY;
	END_CASE

END_FUNCTION

// POUs/EventLogger/getEventClassText
//Returns event class in english and upper case letters 
FUNCTION getEventClassText : STRING(12)
VAR_INPUT
	TcEventClass													: E_TcEventClass;
END_VAR
VAR
END_VAR

CASE TcEventClass OF
TC2_SYSTEM.TCEVENTCLASS_NONE		: GetEventClassText 	:= 'NONE';	
TC2_SYSTEM.TCEVENTCLASS_MESSAGE		: GetEventClassText 	:= 'MESSAGE';	
TC2_SYSTEM.TCEVENTCLASS_HINT		: GetEventClassText 	:= 'HINT';	
TC2_SYSTEM.TCEVENTCLASS_STATEINFO	: GetEventClassText 	:= 'STATEINFO';	
TC2_SYSTEM.TCEVENTCLASS_INSTRUCTION	: GetEventClassText 	:= 'INSTRUCTION';			 										
TC2_SYSTEM.TCEVENTCLASS_WARNING		: GetEventClassText 	:= 'WARNING';	
TC2_SYSTEM.TCEVENTCLASS_MAINTENANCE	: GetEventClassText 	:= 'MAINTENANCE';		 														
TC2_SYSTEM.TCEVENTCLASS_ALARM		: GetEventClassText 	:= 'ALARM';	
TC2_SYSTEM.TCEVENTCLASS_PARAMERROR	: GetEventClassText 	:= 'PARAMERROR';		
ELSE
	GetEventClassText										:= 'UNKNOWN';
END_CASE

END_FUNCTION

// POUs/Fieldbus/CANopen/CANopenMasterDiag
{attribute 'no_check'}
//EL6751 CanOpen Master via EtherCAT
FUNCTION_BLOCK CANopenMasterDiag                   								
VAR_INPUT                   								
	Enable													:	BOOL := TRUE;		//FB will be processed as long as enable is TRUE 
	ConfirmTrig												:	BOOL;               //Resets error with rising edge        								
	SourceId												: 	UDINT :=  103010; 	//Multisource id 
(* Components *)            								
	IO														:	CanOpenMasterIO;
END_VAR                     								
VAR_OUTPUT                  								
	MasterOK												:	BOOL;				//TRUE when Master Device is OK
	FieldOK													:	BOOL;				//TRUE when Field Devices (Slaves) are OK
END_VAR                     	
VAR
(* internal used variables ***********************************************)
	Rx_ErrorCounter											:	USINT := 0;
	Tx_ErrorCounter											: 	USINT := 0;

(* events *********************************************************)
	Event													:	EventHandlingGrp10 := (AutoConfirm	:= FALSE);
	
(* Dummys **********************************************************)
	i														:	INT ;

END_VAR

	(* CanOpen Master Diag Ctrl 					*)
	(************************************************)

(* Work IO *************************************************)
	IO();

(* Events **************************************************)
	IF Event.no[1].Text1 <> IO.Name OR Event.no[1].Text1 <> ''
	THEN
		FOR i := Event.MIN_EVENT TO Event.MAX_EVENT DO
			Event.no[1].Text1								:= IO.Name;
		END_FOR	
	END_IF

(* 
  Bit 0: CAN-Controller is in BUS-OFF
  Bit 1: CAN-Controller warning limit reached
  Bit 2: Rx-Queue overrun
  Bit 3: Hi-Prio Tx-Queue overrun
  Bit 4: Lo-Prio Tx-Queue overrun
  Bit 5: CAN-Send Error
*)
	Event.no[1].Flag 										:= IO.CanState.0;
	Event.no[2].Flag 										:= IO.CanState.1;
	Event.no[3].Flag 										:= IO.CanState.2;   
	Event.no[4].Flag 										:= IO.CanState.3;   
	Event.no[5].Flag 										:= IO.CanState.4; 	
	Event.no[6].Flag 										:= IO.CanState.5;
	
	IF Rx_ErrorCounter <> IO.RXErrorCounter 
	THEN
		Rx_ErrorCounter 									:= IO.RXErrorCounter;
		Event.no[7].Text1 									:= USINT_TO_STRING(Rx_ErrorCounter);
		Event.no[7].Flag									:= TRUE;		
	ELSIF ConfirmTrig
	THEN
		Event.no[7].Flag									:= FALSE;
	END_IF

	IF Tx_ErrorCounter <> IO.TxErrorCounter
	THEN
		Tx_ErrorCounter 									:= IO.TXErrorCounter;
		Event.no[8].Text1 									:= USINT_TO_STRING(Tx_ErrorCounter);
		Event.no[8].Flag									:= TRUE;		
	ELSIF ConfirmTrig
	THEN
		Event.no[8].Flag 									:= FALSE;
	END_IF	

	Event.no[9].Flag 										:= FALSE;
	Event.no[10].Flag 										:= FALSE;	
	
	Event(
		ConfirmTrig := ConfirmTrig,
		Disable		:= NOT Enable,
		SourceId	:= SourceId);
	

(*******************************************************************************************)

END_FUNCTION_BLOCK

// POUs/Fieldbus/CANopen/CANopenMasterIO
{attribute 'no_check'}
//EL6751 CanOpen Master IOs
FUNCTION_BLOCK CANopenMasterIO
VAR_INPUT
END_VAR
VAR_OUTPUT
(* Inputs *)
	AdsAddr											AT %I*	:	AMSADDR;	//Terminal AMS Net Addr.
	AmsNetIdStr												:	T_AmsNetId;	//AmsNetId String
	EcMasterDevId									AT %I*	: 	UINT; 		//Map to EtherCAT Master DevId
	
	Error											AT %I*	:	USINT;		//Rising edge of Error informs that an error occurred during the execution of the Function Block 
	CanState										AT %I*	:	UINT;		//State of Can Bus
	RXErrorCounter									AT %I*	:	USINT;		//Rx error counter of the CAN controller
	TxErrorCounter									AT %I*	:	USINT;		//Tx error counter of the CAN controller
	DiagFlag										AT %I*	:	BOOL;		//Diag Flag of the last configured CANopen slave
	Name													:	STRING(30) := '';
END_VAR                         					
VAR_OUTPUT CONSTANT
END_VAR
VAR
	IOF_GetBoxNameByAddr									:	IOF_GetBoxNameByAddr := (NETID := '', TMOUT := DEFAULT_ADS_TIMEOUT);
END_VAR

(* CANopen master IO diag										             	 		*)
(********************************************************************************)

(* Get name ******************************************************************************)
IF Name = ''
	AND AdsAddr.port <> 0 AND EcMasterDevId <> 0
	OR IOF_GetBoxNameByAddr.BUSY
	OR IOF_GetBoxNameByAddr.START
THEN
	AmsNetIdStr												:= F_CreateAmsNetId(nIds := AdsAddr.netId);
		
	IOF_GetBoxNameByAddr(
		NETID		:=  , (* Local *)
		DEVICEID	:= UINT_TO_UDINT(EcMasterDevId) ,
		BOXADDR		:= AdsAddr.port ,
		START		:= Name = '' AND NOT IOF_GetBoxNameByAddr.BUSY,
		TMOUT		:= ,
		BOXNAME		=> name);
END_IF
(********************************************************************************)

PROPERTY PUBLIC setName : STRING //Set name if device is not an Ethercat terminal
SET
Name := SetName;
END_SET
END_PROPERTY

END_FUNCTION_BLOCK

// POUs/Fieldbus/EAP/EAP_DEVICE_IO
{attribute 'no_check'}
FUNCTION_BLOCK EAP_DEVICE_IO 
VAR_OUTPUT CONSTANT
END_VAR
VAR_INPUT
	{attribute 'displaymode':='hex'}
	DevCtrl				AT %Q*:	UINT;
END_VAR		
VAR_OUTPUT	
	{attribute 'displaymode':='hex'}
	DevState			AT %I*:	UINT;
	
	LinkError				:	BOOL; //0x0001 = Link error
	ResetRequired			:	BOOL; //0x0002 = I/O locked after link error (I/O reset required)
	OutOfSendResources		:	BOOL; //0x0010 = Out of send resources (I/O reset required)
	WatchdogTriggered		:	BOOL; //0x0020 = Watchdog triggered
	EthMiniportNotFound		:	BOOL; //0x0040 = Ethernet driver (miniport) not found
	ResetActive				:	BOOL; //0x0080 = I/O reset active
END_VAR
VAR
END_VAR

	(* IOs 									*)
	(****************************************)

(* Read status *****************************************)
	LinkError				:= DevState.0;
	ResetRequired			:= DevState.1;
	
	OutOfSendResources		:= DevState.4;
	WatchdogTriggered		:= DevState.5;
	EthMiniportNotFound		:= DevState.6;
	ResetActive				:= DevState.7;
(*******************************************************)

END_FUNCTION_BLOCK

// POUs/Fieldbus/EAP/EAP_PUB_SUB_IO
{attribute 'no_check'}
//Publisher/Subscriber IOs
FUNCTION_BLOCK EAP_PUB_SUB_IO 
VAR_OUTPUT CONSTANT
END_VAR
VAR_INPUT
	{attribute 'displaymode':='hex'}
	FrameCtrl									AT %Q*:	UINT;
END_VAR		
VAR_OUTPUT	
	{attribute 'displaymode':='hex'}
	FrameState									AT %I*:	UINT;
	
	NotSentFrameSkipped								: Bool;
	ErrorFrameOversized								: Bool;
	SubscriberMissing								: Bool;
END_VAR
VAR
END_VAR

	(* IOs 									*)
	(****************************************)

(* Read status *****************************************)
	NotSentFrameSkipped						:= FrameState.0;
	ErrorFrameOversized						:= FrameState.1;
	SubscriberMissing						:= FrameState.2;

(*******************************************************)

PROPERTY PUBLIC disableSending : BOOL
GET
disableSending		:= FrameCtrl.1;
END_GET
SET
FrameCtrl.1				:= disableSending;
END_SET
END_PROPERTY

PROPERTY PUBLIC removeDestMacFromARPCache : BOOL
GET
RemoveDestMacFromARPCache		:= FrameCtrl.1;
END_GET
SET
FrameCtrl.1				:= RemoveDestMacFromARPCache;
END_SET
END_PROPERTY

END_FUNCTION_BLOCK

// POUs/Fieldbus/EAP/EAP_PUB_VAR
{attribute 'no_check'}
//Default IOs of a Publisher network variable 
FUNCTION_BLOCK EAP_PUB_VAR 
VAR_OUTPUT CONSTANT
END_VAR
VAR_INPUT
	VarId						AT %Q*:	UINT;
	{attribute 'displaymode':='hex'}
	VarCtrl						AT %Q*:	UINT;
END_VAR		
VAR_OUTPUT	
	{attribute 'displaymode':='hex'}
	VarState					AT %I*:	UINT;
	
	NotSentVarSkipped					:	BOOL;
END_VAR
VAR
END_VAR

	(* IOs 									*)
	(****************************************)

NotSentVarSkipped							:= VarState.0;

PROPERTY PUBLIC disablePublishing : BOOL
GET
disablePublishing		:= VarCtrl.0;
END_GET
SET
VarCtrl.0				:= disablePublishing;
END_SET
END_PROPERTY

END_FUNCTION_BLOCK

// POUs/Fieldbus/EAP/EAP_SUB_VAR
{attribute 'no_check'}
//Default IOs of a Subscriber network variable 
FUNCTION_BLOCK EAP_SUB_VAR 
VAR_OUTPUT CONSTANT
END_VAR
VAR_INPUT
	VarId					AT %Q*:	UINT;	
	{attribute 'displaymode':='hex'}
	VarCtrl					AT %Q*:	UINT;
END_VAR		
VAR_OUTPUT	
	{attribute 'displaymode':='hex'}
	VarState				AT %I*:	UINT;
	Quality					AT %I*:	UINT;//Duration the variable is not refreshed (in 100µs/0.1ms)	
	CycleIndex				AT %I*:	UINT;//Incremented each publisher cycle
	
	QualityLT					 : LTIME;
	QualityLTMax				 : LTIME;
	
	InvalidHashValueReceived		:	BOOL;
	InvalidVarLengthReceived		:	bool;
END_VAR
VAR
END_VAR

	(* IOs 									*)
	(****************************************)

	QualityLT 								:= TO_LTIME(quality * 100000); //Quality in 100µs to ms
	IF QualityLT > QualityLTMax
	THEN
		QualityLTMax						:= QualityLT;
	END_IF
	
	InvalidHashValueReceived				:= VarState.0;
	InvalidVarLengthReceived				:= VarState.1;

PROPERTY PUBLIC ignoreHashValue : BOOL
GET
ignoreHashValue		:= VarCtrl.0;
END_GET
SET
VarCtrl.0				:= ignoreHashValue;
END_SET
END_PROPERTY

END_FUNCTION_BLOCK

// POUs/Fieldbus/EtherCAT/_Components/EcMasterIO
{attribute 'no_check'}
//EtherCAT Master Device IOs
FUNCTION_BLOCK EcMasterIO
VAR CONSTANT
	DELAY_LINK_OK											:	TIME := T#1S;
END_VAR
VAR_OUTPUT CONSTANT
	MIN_FRAMES												:	INT := 0;
	MAX_FRAMES												:	INT := PARAM.ETHERCAT_MASTER_DEV_IO_MAX_FRAMES; 
END_VAR	            							
VAR_INPUT           							                 							
(* Outputs *)       							
	FrmCtrl											AT %Q*	:	ARRAY [MIN_FRAMES..MAX_FRAMES] OF UINT;	//Link to EtherCAT Master "FrmCtrlXXX" under Outputs, e.g. 0x0001 = prevent 1. EtherCAT command from sending (request NOP)
	FrmWcCtrl										AT %Q*	:	ARRAY [MIN_FRAMES..MAX_FRAMES] OF UINT;	//Link to EtherCAT Master "FrmWcCtrlXXX" under Outputs, e.g. 0x0001 = copy data with wrong working counter of 1. EtherCAT command
	                							
	DevCtrl											AT %Q*	:	UINT := 0; //Link to EtherCAT Master "DevCtrl" under Outputs
END_VAR             							
VAR_OUTPUT          							    
	Name													:	STRING(30) := '';
								
	LinkOK_PortA											:	BOOL;		//TRUE when link is OK on port A
	LinkOK_PortB											:	BOOL;		//TRUE when link is OK on port B - Redundancy port 

	{attribute 'displaymode':='hex'}  
	DevState										AT %I*	:	UINT; (*	Link to EtherCAT Master "DevState" under Inputs,
																				0x0001 = Link error
																				0x0002 = I/O locked after link error (I/O reset required)
																				0x0004 = Link error (redundancy adapter)
																				0x0008 = Missing one frame (redundancy mode)
																				0x0010 = Out of send resources (I/O reset required)
																				0x0020 = Watchdog triggered
																				0x0040 = Ethernet driver (miniport) not found
																				0x0080 = I/O reset active
																				0x0100 = At least one device in 'INIT' state
																				0x0200 = At least one device in 'PRE-OP' state
																				0x0400 = At least one device in 'SAFE-OP' state
																				0x0800 = At least one device indicates an error state
																				0x1000 = DC not in sync *)
	DevStateText											:	T_MAXSTRING;		//shows string of device state
	DevStateBits											:	EC_MASTER_DEVICE_STATE;
	DevStateChanged											:	BOOL; //TRUE if device state changed compared to previous cylce								
   	ResetRequired											:	BOOL;		//TRUE when a reset is requested
	MinOneSlaveNotInOP										:	BOOL;		//TRUE when at least one slave is available but not in OP state
    
	NoOfFrames												:	INT;		//No of frames configured
	FrmState										AT %I*	:	ARRAY [MIN_FRAMES..MAX_FRAMES] OF UINT;	//Link to EtherCAT Master "FrmStateXXX" under Inputs, e.g. 0x0001 = 1. EtherCAT command not sent (NOP requested)
	FrmWcState										AT %I*	:	ARRAY [MIN_FRAMES..MAX_FRAMES] OF UINT;	//Link to EtherCAT Master "FrmWcStateXXX" under Inputs, e.g. 0x0001 = wrong working counter of 1. EtherCAT command received
	FrmInputToggle									AT %I*	:	ARRAY [MIN_FRAMES..MAX_FRAMES] OF UINT;	//Link to EtherCAT Master "FrmInputToggleXXX" under Inputs, e.g. 0x0001 = Toggle Bit: 1. EtherCAT command received new inputs
	AllFramesMissing										:	BOOL;		//TRUE if all frames are missing 
	FramesWCState											:	BOOL;		//TRUE if WC state in at least one frame is <> 0
	FramesWcStateChanged									:	BOOL;		//TRUE if WC state of at least one frame changed compared to previous cylce	
	
	SlaveCount										AT %I*	:	UINT;	//Link to EtherCAT Master "SlaveCount" under Inputs, show actual numer of slaves 
	SlaveCount2										AT %I*	:	UINT;	//Link to EtherCAT Master "SlaveCount2" under Inputs, show actual numer of slaves in redunance mode
	SlaveCountTotal											:	UINT; 		//Slave count 1 and 2
	RedundanceActive										:	BOOL;		//Redundance active 		
            																				                    	
(* InfoData *)      	
	ChangeCount										AT %I*	:	UINT;					//Link to EtherCAT Master "ChangeCount" under InfoData, shows how often the image of content has changed
	DevId											AT %I*	:	UINT;					//Link to EtherCAT Master "DevId" under InfoData 
 	AmsNetId										AT %I*	:	ARRAY[0..5] OF BYTE; 	//Link to EtherCAT Master "AmsNetId" under InfoData
	AmsNetIdStr												:	T_AmsNetId;	//EtherCAT Master AmsNetId in string format
	CfgSlaveCount									AT %I*	:	UINT;					////Link to EtherCAT Master "CfgSlaveCount" under InfoData, reports configured no of EtherCAT slaves
         
(* DC timestamp *)
	DCTime													:	T_DCTIME64; // RealtimeTick in DC time 64, refreshed once per cycle*)             					
						
END_VAR

VAR
	MemDevState												:	UINT := 9999;	
	MemFrmWcState											:	ARRAY [MIN_FRAMES..MAX_FRAMES] OF UINT;	

	IOF_GetDeviceName										: 	IOF_GetDeviceName := (TMOUT	:= DEFAULT_ADS_TIMEOUT);
	EcMasterFrameCount										:	FB_EcMasterFrameCount := (tTimeout	:= DEFAULT_ADS_TIMEOUT);
	TON_LinkOK_PortA										:	TON := (PT := DELAY_LINK_OK);
	TON_LinkOK_PortB										:	TON := (PT := DELAY_LINK_OK);
	i														:	INT;
END_VAR

(* EcMaster IOs *)
DevStateChanged												:= DevState <> MemDevState;
IF DevStateChanged
THEN
	DevStateBits.NoError									:= DevState = 0;
	DevStateBits.LinkError 									:= DevState.0;
	DevStateBits.IOLockedAfterLinkError	    				:= DevState.1;
	DevStateBits.LinkErrorRedMode							:= DevState.2;
	DevStateBits.MissingOneFrmInRedMode     				:= DevState.3;
	DevStateBits.OutOfSendResources         				:= DevState.4;
	DevStateBits.WatchdogTriggered 		    				:= DevState.5;
	DevStateBits.EthernetDriverNotFound 					:= DevState.6;
	DevStateBits.IOResetActive 			    				:= DevState.7;
	DevStateBits.AtLeastOneSlaveInINIT      				:= DevState.8;
	DevStateBits.AtLeastOneSlaveInPREOP     				:= DevState.9;
	DevStateBits.AtLeastOneSlaveInSAFEOP    				:= DevState.10;
	DevStateBits.AtLeastOneSlaveInERROR     				:= DevState.11;																
	DevStateBits.DcNotInSync 		        				:= DevState.12;
	DevStateText 											:= F_ConvMasterDevStateToString(DevState);
	ResetRequired 											:= DevStateBits.IOLockedAfterLinkError OR DevStateBits.OutOfSendResources;
	MinOneSlaveNotInOP										:= DevStateBits.AtLeastOneSlaveInINIT OR DevStateBits.AtLeastOneSlaveInPREOP OR  DevStateBits.AtLeastOneSlaveInSAFEOP OR DevStateBits.AtLeastOneSlaveInERROR;
	MemDevState												:= DevState;
END_IF

RedundanceActive 											:= SlaveCount2 <> 0 AND SlaveCount <> 0;
SlaveCountTotal												:= SlaveCount2 + SlaveCount;

TON_LinkOK_PortA(IN:= NOT DevStateBits.LinkError 		, Q=> LinkOK_PortA );
TON_LinkOK_PortB(IN:= NOT DevStateBits.LinkErrorRedMode	, Q=> LinkOK_PortB );

